gfCNCPoint3[10874] = {X 388.1959, Y 11.2433, Z -3.8333, A 0.000, B 0.000, C 0.000 }
gfCNCPoint3[10875] = {X 388.5095, Y 10.3472, Z -3.8333, A 0.000, B 0.000, C 0.000 }
gfCNCPoint3[10876] = {X 389.0147, Y 9.5432, Z -3.8333, A 0.000, B 0.000, C 0.000 }
gfCNCPoint3[10877] = {X 389.6860, Y 8.8719, Z -3.8333, A 0.000, B 0.000, C 0.000 }
gfCNCPoint3[10878] = {X 390.4900, Y 8.3667, Z -3.8333, A 0.000, B 0.000, C 0.000 }
gfCNCPoint3[10879] = {X 391.3861, Y 8.0531, Z -3.8333, A 0.000, B 0.000, C 0.000 }
gfCNCPoint3[10880] = {X 392.3296, Y 7.9468, Z -3.8333, A 0.000, B 0.000, C 0.000 }
gfCNCPoint3[10881] = {X 399.1118, Y 7.9468, Z -3.8333, A 0.000, B 0.000, C 0.000 }
gfCNCPoint3[10882] = {X 400.0552, Y 8.0531, Z -3.8333, A 0.000, B 0.000, C 0.000 }
gfCNCPoint3[10883] = {X 400.9514, Y 8.3667, Z -3.8333, A 0.000, B 0.000, C 0.000 }
gfCNCPoint3[10884] = {X 401.7554, Y 8.8718, Z -3.8333, A 0.000, B 0.000, C 0.000 }
gfCNCPoint3[10885] = {X 402.4267, Y 9.5432, Z -3.8333, A 0.000, B 0.000, C 0.000 }
gfCNCPoint3[10886] = {X 402.9319, Y 10.3471, Z -3.8333, A 0.000, B 0.000, C 0.000 }
gfCNCPoint3[10887] = {X 403.2455, Y 11.2433, Z -3.8333, A 0.000, B 0.000, C 0.000 }
gfCNCPoint3[10888] = {X 403.3518, Y 12.1868, Z -3.8333, A 0.000, B 0.000, C 0.000 }
gfCNCPoint3[10889] = {X 403.3518, Y 12.9781, Z -3.8333, A 0.000, B 0.000, C 0.000 }
gfCNCPoint3[10890] = {X 403.2466, Y 13.9164, Z -3.8333, A 0.000, B 0.000, C 0.000 }
gfCNCPoint3[10891] = {X 402.9365, Y 14.8081, Z -3.8333, A 0.000, B 0.000, C 0.000 }
gfCNCPoint3[10892] = {X 405.3544, Y 18.9789, Z -3.8333, A 0.000, B 0.000, C 0.000 }
gfCNCPoint3[10893] = {X 407.9641, Y 14.7597, Z -3.8333, A 0.000, B 0.000, C 0.000 }
gfCNCPoint3[10894] = {X 407.6748, Y 13.9080, Z -3.8333, A 0.000, B 0.000, C 0.000 }
gfCNCPoint3[10895] = {X 407.5717, Y 13.0144, Z -3.8333, A 0.000, B 0.000, C 0.000 }
gfCNCPoint3[10896] = {X 407.5715, Y 12.1868, Z -3.8333, A 0.000, B 0.000, C 0.000 }
gfCNCPoint3[10897] = {X 407.6778, Y 11.2433, Z -3.8333, A 0.000, B 0.000, C 0.000 }
gfCNCPoint3[10898] = {X 407.9914, Y 10.3471, Z -3.8333, A 0.000, B 0.000, C 0.000 }
gfCNCPoint3[10899] = {X 408.4966, Y 9.5432, Z -3.8333, A 0.000, B 0.000, C 0.000 }
gfCNCPoint3[10900] = {X 409.1679, Y 8.8718, Z -3.8333, A 0.000, B 0.000, C 0.000 }
gfCNCPoint3[10901] = {X 409.9719, Y 8.3667, Z -3.8333, A 0.000, B 0.000, C 0.000 }
gfCNCPoint3[10902] = {X 410.8680, Y 8.0531, Z -3.8333, A 0.000, B 0.000, C 0.000 }
gfCNCPoint3[10903] = {X 411.8115, Y 7.9468, Z -3.8333, A 0.000, B 0.000, C 0.000 }
gfCNCPoint3[10904] = {X 419.3245, Y 7.9468, Z -3.8333, A 0.000, B 0.000, C 0.000 }
gfCNCPoint3[10905] = {X 420.2679, Y 8.0531, Z -3.8333, A 0.000, B 0.000, C 0.000 }
gfCNCPoint3[10906] = {X 421.1641, Y 8.3667, Z -3.8333, A 0.000, B 0.000, C 0.000 }
gfCNCPoint3[10907] = {X 421.9681, Y 8.8718, Z -3.8333, A 0.000, B 0.000, C 0.000 }
gfCNCPoint3[10908] = {X 422.6394, Y 9.5432, Z -3.8333, A 0.000, B 0.000, C 0.000 }
gfCNCPoint3[10909] = {X 423.1446, Y 10.3471, Z -3.8333, A 0.000, B 0.000, C 0.000 }
gfCNCPoint3[10910] = {X 423.4582, Y 11.2433, Z -3.8333, A 0.000, B 0.000, C 0.000 }
gfCNCPoint3[10911] = {X 423.5645, Y 12.1868, Z -3.8333, A 0.000, B 0.000, C 0.000 }
gfCNCPoint3[10912] = {X 423.5645, Y 12.9798, Z -3.8333, A 0.000, B 0.000, C 0.000 }
gfCNCPoint3[10913] = {X 423.4723, Y 13.8340, Z -3.8333, A 0.000, B 0.000, C 0.000 }
gfCNCPoint3[10914] = {X 423.2124, Y 14.6529, Z -3.8333, A 0.000, B 0.000, C 0.000 }
gfCNCPoint3[10915] = {X 422.7950, Y 15.4039, Z -3.8333, A 0.000, B 0.000, C 0.000 }
gfCNCPoint3[10916] = {X 422.2368, Y 16.0570, Z -3.8333, A 0.000, B 0.000, C 0.000 }
gfCNCPoint3[10917] = {X 421.5600, Y 16.5863, Z -3.8333, A 0.000, B 0.000, C 0.000 }
gfCNCPoint3[10918] = {X 420.7916, Y 16.9706, Z -3.8333, A 0.000, B 0.000, C 0.000 }
gfCNCPoint3[10919] = {X 420.0648, Y 17.9463, Z -3.8333, A 0.000, B 0.000, C 0.000 }
gfCNCPoint3[10920] = {X 419.4075, Y 18.9700, Z -3.8333, A 0.000, B 0.000, C 0.000 }
gfCNCPoint3[10921] = {X 417.9262, Y 21.3685, Z -3.8333, A 0.000, B 0.000, C 0.000 }
gfCNCPoint3[10922] = {X 416.0825, Y 24.3294, Z -3.8333, A 0.000, B 0.000, C 0.000 }
gfCNCPoint3[10923] = {X 419.4780, Y 26.4437, Z -3.8333, A 0.000, B 0.000, C 0.000 }
gfCNCPoint3[10924] = {X 416.0146, Y 24.2871, Z -3.8333, A 0.000, B 0.000, C 0.000 }
gfCNCPoint3[10925] = {X 411.3866, Y 31.7193, Z -3.8333, A 0.000, B 0.000, C 0.000 }
gfCNCPoint3[10926] = {X 411.3873, Y 40.9718, Z -3.8333, A 0.000, B 0.000, C 0.000 }
gfCNCPoint3[10927] = {X 412.0246, Y 41.6368, Z -3.8333, A 0.000, B 0.000, C 0.000 }
gfCNCPoint3[10928] = {X 412.5050, Y 42.4226, Z -3.8333, A 0.000, B 0.000, C 0.000 }
gfCNCPoint3[10929] = {X 412.8064, Y 43.2930, Z -3.8333, A 0.000, B 0.000, C 0.000 }
gfCNCPoint3[10930] = {X 412.9147, Y 44.2077, Z -3.8333, A 0.000, B 0.000, C 0.000 }
gfCNCPoint3[10931] = {X 412.9147, Y 45.0002, Z -3.8333, A 0.000, B 0.000, C 0.000 }
gfCNCPoint3[10932] = {X 412.8103, Y 45.9258, Z -3.8333, A 0.000, B 0.000, C 0.000 }
gfCNCPoint3[10933] = {X 412.5027, Y 46.8051, Z -3.8333, A 0.000, B 0.000, C 0.000 }
gfCNCPoint3[10934] = {X 412.0070, Y 47.5938, Z -3.8333, A 0.000, B 0.000, C 0.000 }
gfCNCPoint3[10935] = {X 411.3483, Y 48.2525, Z -3.8333, A 0.000, B 0.000, C 0.000 }
gfCNCPoint3[10936] = {X 410.5596, Y 48.7480, Z -3.8333, A 0.000, B 0.000, C 0.000 }
gfCNCPoint3[10937] = {X 409.6803, Y 49.0557, Z -3.8333, A 0.000, B 0.000, C 0.000 }
gfCNCPoint3[10938] = {X 408.7547, Y 49.1600, Z -3.8333, A 0.000, B 0.000, C 0.000 }
gfCNCPoint3[10939] = {X 402.3112, Y 49.1600, Z -3.8333, A 0.000, B 0.000, C 0.000 }
gfCNCPoint3[10940] = {X 401.3900, Y 49.0567, Z -3.8333, A 0.000, B 0.000, C 0.000 }
gfCNCPoint3[10941] = {X 400.5146, Y 48.7520, Z -3.8333, A 0.000, B 0.000, C 0.000 }
gfCNCPoint3[10942] = {X 399.7283, Y 48.2610, Z -3.8333, A 0.000, B 0.000, C 0.000 }
gfCNCPoint3[10943] = {X 399.0703, Y 47.6081, Z -3.8333, A 0.000, B 0.000, C 0.000 }
gfCNCPoint3[10944] = {X 398.5732, Y 46.8257, Z -3.8333, A 0.000, B 0.000, C 0.000 }
gfCNCPoint3[10945] = {X 398.2617, Y 45.9526, Z -3.8333, A 0.000, B 0.000, C 0.000 }
gfCNCPoint3[10946] = {X 398.1513, Y 45.0322, Z -3.8333, A 0.000, B 0.000, C 0.000 }
gfCNCPoint3[10947] = {X 398.1516, Y 44.1549, Z -3.8333, A 0.000, B 0.000, C 0.000 }
gfCNCPoint3[10948] = {X 398.2616, Y 43.2570, Z -3.8333, A 0.000, B 0.000, C 0.000 }
gfCNCPoint3[10949] = {X 398.5630, Y 42.4041, Z -3.8333, A 0.000, B 0.000, C 0.000 }
gfCNCPoint3[10950] = {X 399.0417, Y 41.6366, Z -3.8333, A 0.000, B 0.000, C 0.000 }
gfCNCPoint3[10951] = {X 399.6750, Y 40.9907, Z -3.8333, A 0.000, B 0.000, C 0.000 }
gfCNCPoint3[10952] = {X 399.6327, Y 31.5567, Z -3.8333, A 0.000, B 0.000, C 0.000 }
gfCNCPoint3[10953] = {X 393.6516, Y 21.1559, Z -3.8333, A 0.000, B 0.000, C 0.000 }
gfCNCPoint3[10954] = {X 392.7632, Y 19.6448, Z -3.8333, A 0.000, B 0.000, C 0.000 }
gfCNCPoint3[10955] = {X 391.8461, Y 18.1509, Z -3.8333, A 0.000, B 0.000, C 0.000 }
gfCNCPoint3[10956] = {X 391.3435, Y 17.4543, Z -3.8333, A 0.000, B 0.000, C 0.000 }
gfCNCPoint3[10957] = {X 390.7552, Y 16.8286, Z -3.8333, A 0.000, B 0.000, C 0.000 }
gfCNCPoint3[10958] = {X 389.9030, Y 16.3569, Z -3.8333, A 0.000, B 0.000, C 0.000 }
gfCNCPoint3[10959] = {X 389.1838, Y 15.7000, Z -3.8333, A 0.000, B 0.000, C 0.000 }
gfCNCPoint3[10960] = {X 388.6371, Y 14.8939, Z -3.8333, A 0.000, B 0.000, C 0.000 }
gfCNCPoint3[10961] = {X 388.2928, Y 13.9828, Z -3.8333, A 0.000, B 0.000, C 0.000 }
gfCNCPoint3[10962] = {X 388.1698, Y 13.0166, Z -3.8333, A 0.000, B 0.000, C 0.000 }
gfCNCPoint3[10963] = {X 388.1696, Y 12.1868, Z -3.8333, A 0.000, B 0.000, C 0.000 }
gfCNCPoint3[10964] = {X 388.2739, Y 11.2611, Z -3.8333, A 0.000, B 0.000, C 0.000 }
gfCNCPoint3[10965] = {X 388.5816, Y 10.3819, Z -3.8333, A 0.000, B 0.000, C 0.000 }
gfCNCPoint3[10966] = {X 389.0772, Y 9.5931, Z -3.8333, A 0.000, B 0.000, C 0.000 }
gfCNCPoint3[10967] = {X 389.7359, Y 8.9344, Z -3.8333, A 0.000, B 0.000, C 0.000 }
gfCNCPoint3[10968] = {X 390.5247, Y 8.4388, Z -3.8333, A 0.000, B 0.000, C 0.000 }
gfCNCPoint3[10969] = {X 391.4039, Y 8.1311, Z -3.8333, A 0.000, B 0.000, C 0.000 }
gfCNCPoint3[10970] = {X 392.3296, Y 8.0268, Z -3.8333, A 0.000, B 0.000, C 0.000 }
gfCNCPoint3[10971] = {X 399.1118, Y 8.0268, Z -3.8333, A 0.000, B 0.000, C 0.000 }
gfCNCPoint3[10972] = {X 400.0374, Y 8.1311, Z -3.8333, A 0.000, B 0.000, C 0.000 }
gfCNCPoint3[10973] = {X 400.9167, Y 8.4388, Z -3.8333, A 0.000, B 0.000, C 0.000 }
gfCNCPoint3[10974] = {X 401.7055, Y 8.9344, Z -3.8333, A 0.000, B 0.000, C 0.000 }
gfCNCPoint3[10975] = {X 402.3642, Y 9.5931, Z -3.8333, A 0.000, B 0.000, C 0.000 }
gfCNCPoint3[10976] = {X 402.8598, Y 10.3819, Z -3.8333, A 0.000, B 0.000, C 0.000 }
gfCNCPoint3[10977] = {X 403.1675, Y 11.2611, Z -3.8333, A 0.000, B 0.000, C 0.000 }
gfCNCPoint3[10978] = {X 403.2718, Y 12.1868, Z -3.8333, A 0.000, B 0.000, C 0.000 }
gfCNCPoint3[10979] = {X 403.2718, Y 12.9781, Z -3.8333, A 0.000, B 0.000, C 0.000 }
gfCNCPoint3[10980] = {X 403.1639, Y 13.9192, Z -3.8333, A 0.000, B 0.000, C 0.000 }
gfCNCPoint3[10981] = {X 402.8459, Y 14.8115, Z -3.8333, A 0.000, B 0.000, C 0.000 }
gfCNCPoint3[10982] = {X 405.3522, Y 19.1346, Z -3.8333, A 0.000, B 0.000, C 0.000 }
gfCNCPoint3[10983] = {X 408.0549, Y 14.7650, Z -3.8333, A 0.000, B 0.000, C 0.000 }
gfCNCPoint3[10984] = {X 407.7576, Y 13.9114, Z -3.8333, A 0.000, B 0.000, C 0.000 }
gfCNCPoint3[10985] = {X 407.6517, Y 13.0137, Z -3.8333, A 0.000, B 0.000, C 0.000 }
gfCNCPoint3[10986] = {X 407.6515, Y 12.1868, Z -3.8333, A 0.000, B 0.000, C 0.000 }
gfCNCPoint3[10987] = {X 407.7558, Y 11.2611, Z -3.8333, A 0.000, B 0.000, C 0.000 }
gfCNCPoint3[10988] = {X 408.0635, Y 10.3819, Z -3.8333, A 0.000, B 0.000, C 0.000 }
gfCNCPoint3[10989] = {X 408.5591, Y 9.5931, Z -3.8333, A 0.000, B 0.000, C 0.000 }
gfCNCPoint3[10990] = {X 409.2178, Y 8.9344, Z -3.8333, A 0.000, B 0.000, C 0.000 }
gfCNCPoint3[10991] = {X 410.0066, Y 8.4388, Z -3.8333, A 0.000, B 0.000, C 0.000 }
gfCNCPoint3[10992] = {X 410.8859, Y 8.1311, Z -3.8333, A 0.000, B 0.000, C 0.000 }
gfCNCPoint3[10993] = {X 411.8115, Y 8.0268, Z -3.8333, A 0.000, B 0.000, C 0.000 }
gfCNCPoint3[10994] = {X 419.3245, Y 8.0268, Z -3.8333, A 0.000, B 0.000, C 0.000 }
gfCNCPoint3[10995] = {X 420.2501, Y 8.1311, Z -3.8333, A 0.000, B 0.000, C 0.000 }
gfCNCPoint3[10996] = {X 421.1294, Y 8.4388, Z -3.8333, A 0.000, B 0.000, C 0.000 }
gfCNCPoint3[10997] = {X 421.9182, Y 8.9344, Z -3.8333, A 0.000, B 0.000, C 0.000 }
gfCNCPoint3[10998] = {X 422.5769, Y 9.5931, Z -3.8333, A 0.000, B 0.000, C 0.000 }
gfCNCPoint3[10999] = {X 423.0725, Y 10.3819, Z -3.8333, A 0.000, B 0.000, C 0.000 }
gfCNCPoint3[11000] = {X 423.3802, Y 11.2611, Z -3.8333, A 0.000, B 0.000, C 0.000 }
gfCNCPoint3[11001] = {X 423.4845, Y 12.1868, Z -3.8333, A 0.000, B 0.000, C 0.000 }
gfCNCPoint3[11002] = {X 423.4845, Y 12.9792, Z -3.8333, A 0.000, B 0.000, C 0.000 }
gfCNCPoint3[11003] = {X 423.3933, Y 13.8210, Z -3.8333, A 0.000, B 0.000, C 0.000 }
gfCNCPoint3[11004] = {X 423.1361, Y 14.6278, Z -3.8333, A 0.000, B 0.000, C 0.000 }
gfCNCPoint3[11005] = {X 422.7231, Y 15.3671, Z -3.8333, A 0.000, B 0.000, C 0.000 }
gfCNCPoint3[11006] = {X 422.1710, Y 16.0092, Z -3.8333, A 0.000, B 0.000, C 0.000 }
gfCNCPoint3[11007] = {X 421.5020, Y 16.5283, Z -3.8333, A 0.000, B 0.000, C 0.000 }
gfCNCPoint3[11008] = {X 420.7429, Y 16.9035, Z -3.8333, A 0.000, B 0.000, C 0.000 }
gfCNCPoint3[11009] = {X 420.0054, Y 17.8914, Z -3.8333, A 0.000, B 0.000, C 0.000 }
gfCNCPoint3[11010] = {X 419.3390, Y 18.9286, Z -3.8333, A 0.000, B 0.000, C 0.000 }
gfCNCPoint3[11011] = {X 417.8583, Y 21.3264, Z -3.8333, A 0.000, B 0.000, C 0.000 }
gfCNCPoint3[11012] = {X 416.0146, Y 24.2871, Z -3.8333, A 0.000, B 0.000, C 0.000 }
gfCNCPoint3[11013] = {X 419.4101, Y 26.4014, Z -3.8333, A 0.000, B 0.000, C 0.000 }
gfCNCPoint3[11014] = {X 415.9467, Y 24.2448, Z -3.8333, A 0.000, B 0.000, C 0.000 }
gfCNCPoint3[11015] = {X 411.3066, Y 31.6964, Z -3.8333, A 0.000, B 0.000, C 0.000 }
gfCNCPoint3[11016] = {X 411.3073, Y 41.0093, Z -3.8333, A 0.000, B 0.000, C 0.000 }
gfCNCPoint3[11017] = {X 411.9442, Y 41.6636, Z -3.8333, A 0.000, B 0.000, C 0.000 }
gfCNCPoint3[11018] = {X 412.4247, Y 42.4400, Z -3.8333, A 0.000, B 0.000, C 0.000 }
gfCNCPoint3[11019] = {X 412.7263, Y 43.3018, Z -3.8333, A 0.000, B 0.000, C 0.000 }
gfCNCPoint3[11020] = {X 412.8347, Y 44.2085, Z -3.8333, A 0.000, B 0.000, C 0.000 }
gfCNCPoint3[11021] = {X 412.8347, Y 45.0002, Z -3.8333, A 0.000, B 0.000, C 0.000 }
gfCNCPoint3[11022] = {X 412.7324, Y 45.9080, Z -3.8333, A 0.000, B 0.000, C 0.000 }
gfCNCPoint3[11023] = {X 412.4306, Y 46.7703, Z -3.8333, A 0.000, B 0.000, C 0.000 }
gfCNCPoint3[11024] = {X 411.9445, Y 47.5439, Z -3.8333, A 0.000, B 0.000, C 0.000 }
gfCNCPoint3[11025] = {X 411.2985, Y 48.1899, Z -3.8333, A 0.000, B 0.000, C 0.000 }
gfCNCPoint3[11026] = {X 410.5249, Y 48.6760, Z -3.8333, A 0.000, B 0.000, C 0.000 }
gfCNCPoint3[11027] = {X 409.6625, Y 48.9777, Z -3.8333, A 0.000, B 0.000, C 0.000 }
gfCNCPoint3[11028] = {X 408.7547, Y 49.0800, Z -3.8333, A 0.000, B 0.000, C 0.000 }
gfCNCPoint3[11029] = {X 402.3112, Y 49.0800, Z -3.8333, A 0.000, B 0.000, C 0.000 }
gfCNCPoint3[11030] = {X 401.4077, Y 48.9787, Z -3.8333, A 0.000, B 0.000, C 0.000 }
gfCNCPoint3[11031] = {X 400.5491, Y 48.6799, Z -3.8333, A 0.000, B 0.000, C 0.000 }
gfCNCPoint3[11032] = {X 399.7780, Y 48.1983, Z -3.8333, A 0.000, B 0.000, C 0.000 }
gfCNCPoint3[11033] = {X 399.1326, Y 47.5579, Z -3.8333, A 0.000, B 0.000, C 0.000 }
gfCNCPoint3[11034] = {X 398.6451, Y 46.7906, Z -3.8333, A 0.000, B 0.000, C 0.000 }
gfCNCPoint3[11035] = {X 398.3396, Y 45.9343, Z -3.8333, A 0.000, B 0.000, C 0.000 }
gfCNCPoint3[11036] = {X 398.2313, Y 45.0316, Z -3.8333, A 0.000, B 0.000, C 0.000 }
gfCNCPoint3[11037] = {X 398.2316, Y 44.1559, Z -3.8333, A 0.000, B 0.000, C 0.000 }
gfCNCPoint3[11038] = {X 398.3416, Y 43.2661, Z -3.8333, A 0.000, B 0.000, C 0.000 }
gfCNCPoint3[11039] = {X 398.6434, Y 42.4218, Z -3.8333, A 0.000, B 0.000, C 0.000 }
gfCNCPoint3[11040] = {X 399.1223, Y 41.6638, Z -3.8333, A 0.000, B 0.000, C 0.000 }
gfCNCPoint3[11041] = {X 399.7552, Y 41.0287, Z -3.8333, A 0.000, B 0.000, C 0.000 }
gfCNCPoint3[11042] = {X 399.7126, Y 31.5351, Z -3.8333, A 0.000, B 0.000, C 0.000 }
gfCNCPoint3[11043] = {X 393.7210, Y 21.1161, Z -3.8333, A 0.000, B 0.000, C 0.000 }
gfCNCPoint3[11044] = {X 392.8318, Y 19.6036, Z -3.8333, A 0.000, B 0.000, C 0.000 }
gfCNCPoint3[11045] = {X 391.9139, Y 18.1084, Z -3.8333, A 0.000, B 0.000, C 0.000 }
gfCNCPoint3[11046] = {X 391.4005, Y 17.3977, Z -3.8333, A 0.000, B 0.000, C 0.000 }
gfCNCPoint3[11047] = {X 390.7990, Y 16.7600, Z -3.8333, A 0.000, B 0.000, C 0.000 }
gfCNCPoint3[11048] = {X 389.9591, Y 16.2987, Z -3.8333, A 0.000, B 0.000, C 0.000 }
gfCNCPoint3[11049] = {X 389.2500, Y 15.6543, Z -3.8333, A 0.000, B 0.000, C 0.000 }
gfCNCPoint3[11050] = {X 388.7108, Y 14.8623, Z -3.8333, A 0.000, B 0.000, C 0.000 }
gfCNCPoint3[11051] = {X 388.3711, Y 13.9663, Z -3.8333, A 0.000, B 0.000, C 0.000 }
gfCNCPoint3[11052] = {X 388.2498, Y 13.0158, Z -3.8333, A 0.000, B 0.000, C 0.000 }
gfCNCPoint3[11053] = {X 388.2496, Y 12.1868, Z -3.8333, A 0.000, B 0.000, C 0.000 }
gfCNCPoint3[11054] = {X 388.3519, Y 11.2789, Z -3.8333, A 0.000, B 0.000, C 0.000 }
gfCNCPoint3[11055] = {X 388.6537, Y 10.4166, Z -3.8333, A 0.000, B 0.000, C 0.000 }
gfCNCPoint3[11056] = {X 389.1398, Y 9.6430, Z -3.8333, A 0.000, B 0.000, C 0.000 }
gfCNCPoint3[11057] = {X 389.7858, Y 8.9969, Z -3.8333, A 0.000, B 0.000, C 0.000 }
gfCNCPoint3[11058] = {X 390.5594, Y 8.5109, Z -3.8333, A 0.000, B 0.000, C 0.000 }
gfCNCPoint3[11059] = {X 391.4217, Y 8.2091, Z -3.8333, A 0.000, B 0.000, C 0.000 }
gfCNCPoint3[11060] = {X 392.3296, Y 8.1068, Z -3.8333, A 0.000, B 0.000, C 0.000 }
gfCNCPoint3[11061] = {X 399.1118, Y 8.1068, Z -3.8333, A 0.000, B 0.000, C 0.000 }
gfCNCPoint3[11062] = {X 400.0196, Y 8.2091, Z -3.8333, A 0.000, B 0.000, C 0.000 }
gfCNCPoint3[11063] = {X 400.8820, Y 8.5109, Z -3.8333, A 0.000, B 0.000, C 0.000 }
gfCNCPoint3[11064] = {X 401.6556, Y 8.9969, Z -3.8333, A 0.000, B 0.000, C 0.000 }
gfCNCPoint3[11065] = {X 402.3016, Y 9.6430, Z -3.8333, A 0.000, B 0.000, C 0.000 }
gfCNCPoint3[11066] = {X 402.7877, Y 10.4166, Z -3.8333, A 0.000, B 0.000, C 0.000 }
gfCNCPoint3[11067] = {X 403.0895, Y 11.2789, Z -3.8333, A 0.000, B 0.000, C 0.000 }
gfCNCPoint3[11068] = {X 403.1918, Y 12.1868, Z -3.8333, A 0.000, B 0.000, C 0.000 }
gfCNCPoint3[11069] = {X 403.1918, Y 12.9781, Z -3.8333, A 0.000, B 0.000, C 0.000 }
gfCNCPoint3[11070] = {X 403.0811, Y 13.9219, Z -3.8333, A 0.000, B 0.000, C 0.000 }
gfCNCPoint3[11071] = {X 402.7551, Y 14.8144, Z -3.8333, A 0.000, B 0.000, C 0.000 }
gfCNCPoint3[11072] = {X 405.3499, Y 19.2903, Z -3.8333, A 0.000, B 0.000, C 0.000 }
gfCNCPoint3[11073] = {X 408.1460, Y 14.7697, Z -3.8333, A 0.000, B 0.000, C 0.000 }
gfCNCPoint3[11074] = {X 408.1093, Y 14.6926, Z -3.8333, A 0.000, B 0.000, C 0.000 }
gfCNCPoint3[11075] = {X 408.0742, Y 14.6147, Z -3.8333, A 0.000, B 0.000, C 0.000 }
gfCNCPoint3[11076] = {X 407.8218, Y 13.8313, Z -3.8333, A 0.000, B 0.000, C 0.000 }
gfCNCPoint3[11077] = {X 407.7317, Y 13.0131, Z -3.8333, A 0.000, B 0.000, C 0.000 }
gfCNCPoint3[11078] = {X 407.7315, Y 12.1868, Z -3.8333, A 0.000, B 0.000, C 0.000 }
gfCNCPoint3[11079] = {X 407.8338, Y 11.2789, Z -3.8333, A 0.000, B 0.000, C 0.000 }
gfCNCPoint3[11080] = {X 408.1356, Y 10.4166, Z -3.8333, A 0.000, B 0.000, C 0.000 }
gfCNCPoint3[11081] = {X 408.6217, Y 9.6430, Z -3.8333, A 0.000, B 0.000, C 0.000 }
gfCNCPoint3[11082] = {X 409.2677, Y 8.9969, Z -3.8333, A 0.000, B 0.000, C 0.000 }
gfCNCPoint3[11083] = {X 410.0413, Y 8.5109, Z -3.8333, A 0.000, B 0.000, C 0.000 }
gfCNCPoint3[11084] = {X 410.9037, Y 8.2091, Z -3.8333, A 0.000, B 0.000, C 0.000 }
gfCNCPoint3[11085] = {X 411.8115, Y 8.1068, Z -3.8333, A 0.000, B 0.000, C 0.000 }
gfCNCPoint3[11086] = {X 419.3245, Y 8.1068, Z -3.8333, A 0.000, B 0.000, C 0.000 }
gfCNCPoint3[11087] = {X 420.2323, Y 8.2091, Z -3.8333, A 0.000, B 0.000, C 0.000 }
gfCNCPoint3[11088] = {X 421.0947, Y 8.5109, Z -3.8333, A 0.000, B 0.000, C 0.000 }
gfCNCPoint3[11089] = {X 421.8683, Y 8.9969, Z -3.8333, A 0.000, B 0.000, C 0.000 }
gfCNCPoint3[11090] = {X 422.5143, Y 9.6430, Z -3.8333, A 0.000, B 0.000, C 0.000 }
gfCNCPoint3[11091] = {X 423.0004, Y 10.4166, Z -3.8333, A 0.000, B 0.000, C 0.000 }
gfCNCPoint3[11092] = {X 423.3022, Y 11.2789, Z -3.8333, A 0.000, B 0.000, C 0.000 }
gfCNCPoint3[11093] = {X 423.4045, Y 12.1868, Z -3.8333, A 0.000, B 0.000, C 0.000 }
gfCNCPoint3[11094] = {X 423.4045, Y 12.9786, Z -3.8333, A 0.000, B 0.000, C 0.000 }
gfCNCPoint3[11095] = {X 423.3143, Y 13.8081, Z -3.8333, A 0.000, B 0.000, C 0.000 }
gfCNCPoint3[11096] = {X 423.0598, Y 14.6027, Z -3.8333, A 0.000, B 0.000, C 0.000 }
gfCNCPoint3[11097] = {X 422.6513, Y 15.3302, Z -3.8333, A 0.000, B 0.000, C 0.000 }
gfCNCPoint3[11098] = {X 422.1053, Y 15.9612, Z -3.8333, A 0.000, B 0.000, C 0.000 }
gfCNCPoint3[11099] = {X 421.4441, Y 16.4701, Z -3.8333, A 0.000, B 0.000, C 0.000 }
gfCNCPoint3[11100] = {X 420.6943, Y 16.8362, Z -3.8333, A 0.000, B 0.000, C 0.000 }
gfCNCPoint3[11101] = {X 419.9462, Y 17.8365, Z -3.8333, A 0.000, B 0.000, C 0.000 }
gfCNCPoint3[11102] = {X 419.2706, Y 18.8871, Z -3.8333, A 0.000, B 0.000, C 0.000 }
gfCNCPoint3[11103] = {X 417.7903, Y 21.2842, Z -3.8333, A 0.000, B 0.000, C 0.000 }
gfCNCPoint3[11104] = {X 415.9467, Y 24.2448, Z -3.8333, A 0.000, B 0.000, C 0.000 }
gfCNCPoint3[11105] = {X 419.3422, Y 26.3592, Z -3.8333, A 0.000, B 0.000, C 0.000 }
gfCNCPoint3[11106] = {X 415.8788, Y 24.2025, Z -3.8333, A 0.000, B 0.000, C 0.000 }
gfCNCPoint3[11107] = {X 411.2266, Y 31.6735, Z -3.8333, A 0.000, B 0.000, C 0.000 }
gfCNCPoint3[11108] = {X 411.2273, Y 41.0472, Z -3.8333, A 0.000, B 0.000, C 0.000 }
gfCNCPoint3[11109] = {X 411.8636, Y 41.6906, Z -3.8333, A 0.000, B 0.000, C 0.000 }
gfCNCPoint3[11110] = {X 412.3443, Y 42.4574, Z -3.8333, A 0.000, B 0.000, C 0.000 }
gfCNCPoint3[11111] = {X 412.6462, Y 43.3105, Z -3.8333, A 0.000, B 0.000, C 0.000 }
gfCNCPoint3[11112] = {X 412.7547, Y 44.2089, Z -3.8333, A 0.000, B 0.000, C 0.000 }
gfCNCPoint3[11113] = {X 412.7545, Y 45.0384, Z -3.8333, A 0.000, B 0.000, C 0.000 }
gfCNCPoint3[11114] = {X 412.6469, Y 45.9222, Z -3.8333, A 0.000, B 0.000, C 0.000 }
gfCNCPoint3[11115] = {X 412.3466, Y 46.7602, Z -3.8333, A 0.000, B 0.000, C 0.000 }
gfCNCPoint3[11116] = {X 411.8683, Y 47.5111, Z -3.8333, A 0.000, B 0.000, C 0.000 }
gfCNCPoint3[11117] = {X 411.2357, Y 48.1376, Z -3.8333, A 0.000, B 0.000, C 0.000 }
gfCNCPoint3[11118] = {X 410.4803, Y 48.6086, Z -3.8333, A 0.000, B 0.000, C 0.000 }
gfCNCPoint3[11119] = {X 409.6394, Y 48.9009, Z -3.8333, A 0.000, B 0.000, C 0.000 }
gfCNCPoint3[11120] = {X 408.7547, Y 49.0000, Z -3.8333, A 0.000, B 0.000, C 0.000 }
gfCNCPoint3[11121] = {X 402.3112, Y 49.0000, Z -3.8333, A 0.000, B 0.000, C 0.000 }
gfCNCPoint3[11122] = {X 401.4211, Y 48.8997, Z -3.8333, A 0.000, B 0.000, C 0.000 }
gfCNCPoint3[11123] = {X 400.5757, Y 48.6039, Z -3.8333, A 0.000, B 0.000, C 0.000 }
gfCNCPoint3[11124] = {X 399.8172, Y 48.1273, Z -3.8333, A 0.000, B 0.000, C 0.000 }
gfCNCPoint3[11125] = {X 399.1839, Y 47.4939, Z -3.8333, A 0.000, B 0.000, C 0.000 }
gfCNCPoint3[11126] = {X 398.7073, Y 46.7355, Z -3.8333, A 0.000, B 0.000, C 0.000 }
gfCNCPoint3[11127] = {X 398.4115, Y 45.8900, Z -3.8333, A 0.000, B 0.000, C 0.000 }
gfCNCPoint3[11128] = {X 398.3112, Y 45.0000, Z -3.8333, A 0.000, B 0.000, C 0.000 }
gfCNCPoint3[11129] = {X 398.3115, Y 44.1569, Z -3.8333, A 0.000, B 0.000, C 0.000 }
gfCNCPoint3[11130] = {X 398.4217, Y 43.2753, Z -3.8333, A 0.000, B 0.000, C 0.000 }
gfCNCPoint3[11131] = {X 398.7237, Y 42.4397, Z -3.8333, A 0.000, B 0.000, C 0.000 }
gfCNCPoint3[11132] = {X 399.2028, Y 41.6913, Z -3.8333, A 0.000, B 0.000, C 0.000 }
gfCNCPoint3[11133] = {X 399.8352, Y 41.0672, Z -3.8333, A 0.000, B 0.000, C 0.000 }
gfCNCPoint3[11134] = {X 399.8376, Y 31.5921, Z -3.8333, A 0.000, B 0.000, C 0.000 }
gfCNCPoint3[11135] = {X 393.7903, Y 21.0762, Z -3.8333, A 0.000, B 0.000, C 0.000 }
gfCNCPoint3[11136] = {X 392.9004, Y 19.5624, Z -3.8333, A 0.000, B 0.000, C 0.000 }
gfCNCPoint3[11137] = {X 391.9816, Y 18.0659, Z -3.8333, A 0.000, B 0.000, C 0.000 }
gfCNCPoint3[11138] = {X 391.4575, Y 17.3410, Z -3.8333, A 0.000, B 0.000, C 0.000 }
gfCNCPoint3[11139] = {X 390.8426, Y 16.6913, Z -3.8333, A 0.000, B 0.000, C 0.000 }
gfCNCPoint3[11140] = {X 390.0091, Y 16.2361, Z -3.8333, A 0.000, B 0.000, C 0.000 }
gfCNCPoint3[11141] = {X 389.3064, Y 15.5972, Z -3.8333, A 0.000, B 0.000, C 0.000 }
gfCNCPoint3[11142] = {X 388.7742, Y 14.8107, Z -3.8333, A 0.000, B 0.000, C 0.000 }
gfCNCPoint3[11143] = {X 388.4423, Y 13.9209, Z -3.8333, A 0.000, B 0.000, C 0.000 }
gfCNCPoint3[11144] = {X 388.3296, Y 12.9779, Z -3.8333, A 0.000, B 0.000, C 0.000 }
gfCNCPoint3[11145] = {X 388.3296, Y 12.1868, Z -3.8333, A 0.000, B 0.000, C 0.000 }
gfCNCPoint3[11146] = {X 388.4299, Y 11.2967, Z -3.8333, A 0.000, B 0.000, C 0.000 }
gfCNCPoint3[11147] = {X 388.7258, Y 10.4513, Z -3.8333, A 0.000, B 0.000, C 0.000 }
gfCNCPoint3[11148] = {X 389.2023, Y 9.6929, Z -3.8333, A 0.000, B 0.000, C 0.000 }
gfCNCPoint3[11149] = {X 389.8357, Y 9.0595, Z -3.8333, A 0.000, B 0.000, C 0.000 }
gfCNCPoint3[11150] = {X 390.5941, Y 8.5829, Z -3.8333, A 0.000, B 0.000, C 0.000 }
gfCNCPoint3[11151] = {X 391.4395, Y 8.2871, Z -3.8333, A 0.000, B 0.000, C 0.000 }
gfCNCPoint3[11152] = {X 392.3296, Y 8.1868, Z -3.8333, A 0.000, B 0.000, C 0.000 }
gfCNCPoint3[11153] = {X 399.1118, Y 8.1868, Z -3.8333, A 0.000, B 0.000, C 0.000 }
gfCNCPoint3[11154] = {X 400.0018, Y 8.2871, Z -3.8333, A 0.000, B 0.000, C 0.000 }
gfCNCPoint3[11155] = {X 400.8473, Y 8.5829, Z -3.8333, A 0.000, B 0.000, C 0.000 }
gfCNCPoint3[11156] = {X 401.6057, Y 9.0595, Z -3.8333, A 0.000, B 0.000, C 0.000 }
gfCNCPoint3[11157] = {X 402.2391, Y 9.6929, Z -3.8333, A 0.000, B 0.000, C 0.000 }
gfCNCPoint3[11158] = {X 402.7156, Y 10.4513, Z -3.8333, A 0.000, B 0.000, C 0.000 }
gfCNCPoint3[11159] = {X 403.0115, Y 11.2967, Z -3.8333, A 0.000, B 0.000, C 0.000 }
gfCNCPoint3[11160] = {X 403.1118, Y 12.1868, Z -3.8333, A 0.000, B 0.000, C 0.000 }
gfCNCPoint3[11161] = {X 403.1115, Y 13.0192, Z -3.8333, A 0.000, B 0.000, C 0.000 }
gfCNCPoint3[11162] = {X 402.9933, Y 13.9442, Z -3.8333, A 0.000, B 0.000, C 0.000 }
gfCNCPoint3[11163] = {X 402.6641, Y 14.8167, Z -3.8333, A 0.000, B 0.000, C 0.000 }
gfCNCPoint3[11164] = {X 405.2576, Y 19.3199, Z -3.8333, A 0.000, B 0.000, C 0.000 }
gfCNCPoint3[11165] = {X 405.3712, Y 19.4080, Z -3.8333, A 0.000, B 0.000, C 0.000 }
gfCNCPoint3[11166] = {X 408.1949, Y 14.8342, Z -3.8333, A 0.000, B 0.000, C 0.000 }
gfCNCPoint3[11167] = {X 408.2428, Y 14.7847, Z -3.8333, A 0.000, B 0.000, C 0.000 }
gfCNCPoint3[11168] = {X 408.1937, Y 14.6843, Z -3.8333, A 0.000, B 0.000, C 0.000 }
gfCNCPoint3[11169] = {X 408.1475, Y 14.5826, Z -3.8333, A 0.000, B 0.000, C 0.000 }
gfCNCPoint3[11170] = {X 407.8964, Y 13.7977, Z -3.8333, A 0.000, B 0.000, C 0.000 }
gfCNCPoint3[11171] = {X 407.8115, Y 12.9779, Z -3.8333, A 0.000, B 0.000, C 0.000 }
gfCNCPoint3[11172] = {X 407.8115, Y 12.1868, Z -3.8333, A 0.000, B 0.000, C 0.000 }
gfCNCPoint3[11173] = {X 407.9118, Y 11.2967, Z -3.8333, A 0.000, B 0.000, C 0.000 }
gfCNCPoint3[11174] = {X 408.2077, Y 10.4513, Z -3.8333, A 0.000, B 0.000, C 0.000 }
gfCNCPoint3[11175] = {X 408.6842, Y 9.6929, Z -3.8333, A 0.000, B 0.000, C 0.000 }
gfCNCPoint3[11176] = {X 409.3176, Y 9.0595, Z -3.8333, A 0.000, B 0.000, C 0.000 }
gfCNCPoint3[11177] = {X 410.0760, Y 8.5829, Z -3.8333, A 0.000, B 0.000, C 0.000 }
gfCNCPoint3[11178] = {X 410.9215, Y 8.2871, Z -3.8333, A 0.000, B 0.000, C 0.000 }
gfCNCPoint3[11179] = {X 411.8115, Y 8.1868, Z -3.8333, A 0.000, B 0.000, C 0.000 }
gfCNCPoint3[11180] = {X 419.3245, Y 8.1868, Z -3.8333, A 0.000, B 0.000, C 0.000 }
gfCNCPoint3[11181] = {X 420.2145, Y 8.2871, Z -3.8333, A 0.000, B 0.000, C 0.000 }
gfCNCPoint3[11182] = {X 421.0600, Y 8.5829, Z -3.8333, A 0.000, B 0.000, C 0.000 }
gfCNCPoint3[11183] = {X 421.8184, Y 9.0595, Z -3.8333, A 0.000, B 0.000, C 0.000 }
gfCNCPoint3[11184] = {X 422.4518, Y 9.6929, Z -3.8333, A 0.000, B 0.000, C 0.000 }
gfCNCPoint3[11185] = {X 422.9283, Y 10.4513, Z -3.8333, A 0.000, B 0.000, C 0.000 }
gfCNCPoint3[11186] = {X 423.2242, Y 11.2967, Z -3.8333, A 0.000, B 0.000, C 0.000 }
gfCNCPoint3[11187] = {X 423.3245, Y 12.1868, Z -3.8333, A 0.000, B 0.000, C 0.000 }
gfCNCPoint3[11188] = {X 423.3245, Y 12.9780, Z -3.8333, A 0.000, B 0.000, C 0.000 }
gfCNCPoint3[11189] = {X 423.1977, Y 13.9553, Z -3.8333, A 0.000, B 0.000, C 0.000 }
gfCNCPoint3[11190] = {X 422.8393, Y 14.8735, Z -3.8333, A 0.000, B 0.000, C 0.000 }
gfCNCPoint3[11191] = {X 422.2706, Y 15.6784, Z -3.8333, A 0.000, B 0.000, C 0.000 }
gfCNCPoint3[11192] = {X 421.5249, Y 16.3228, Z -3.8333, A 0.000, B 0.000, C 0.000 }
gfCNCPoint3[11193] = {X 420.6460, Y 16.7687, Z -3.8333, A 0.000, B 0.000, C 0.000 }
gfCNCPoint3[11194] = {X 419.8870, Y 17.7815, Z -3.8333, A 0.000, B 0.000, C 0.000 }
gfCNCPoint3[11195] = {X 419.2022, Y 18.8457, Z -3.8333, A 0.000, B 0.000, C 0.000 }
gfCNCPoint3[11196] = {X 417.7223, Y 21.2420, Z -3.8333, A 0.000, B 0.000, C 0.000 }
gfCNCPoint3[11197] = {X 415.8788, Y 24.2025, Z -3.8333, A 0.000, B 0.000, C 0.000 }
gfCNCPoint3[11198] = {X 419.3422, Y 26.3592, Z -3.8333, A 0.000, B 0.000, C 0.000 }
gfCNCPoint3[11199] = {X 419.3422, Y 26.3592, Z -0.8333, A 0.000, B 0.000, C 0.000 }
gfCNCPoint3[11200] = {X 419.3422, Y 26.3592, Z 11.0000, A 0.000, B 0.000, C 0.000 }
gfCNCPoint3[11201] = {X 352.3320, Y -3.5327, Z 11.0000, A 0.000, B 0.000, C 0.000 }
gfCNCPoint3[11202] = {X 352.3320, Y -3.5327, Z -0.8333, A 0.000, B 0.000, C 0.000 }
gfCNCPoint3[11203] = {X 352.3320, Y -3.5327, Z -3.8333, A 0.000, B 0.000, C 0.000 }
gfCNCPoint3[11204] = {X 351.5861, Y 0.4785, Z -3.8333, A 0.000, B 0.000, C 0.000 }
gfCNCPoint3[11205] = {X 351.8696, Y 0.5313, Z -3.8333, A 0.000, B 0.000, C 0.000 }
gfCNCPoint3[11206] = {X 353.8045, Y 1.0172, Z -3.8333, A 0.000, B 0.000, C 0.000 }
gfCNCPoint3[11207] = {X 355.6846, Y 1.6844, Z -3.8333, A 0.000, B 0.000, C 0.000 }
gfCNCPoint3[11208] = {X 357.4930, Y 2.5269, Z -3.8333, A 0.000, B 0.000, C 0.000 }
gfCNCPoint3[11209] = {X 359.2134, Y 3.5369, Z -3.8333, A 0.000, B 0.000, C 0.000 }
gfCNCPoint3[11210] = {X 360.8303, Y 4.7055, Z -3.8333, A 0.000, B 0.000, C 0.000 }
gfCNCPoint3[11211] = {X 362.3292, Y 6.0221, Z -3.8333, A 0.000, B 0.000, C 0.000 }
gfCNCPoint3[11212] = {X 363.6965, Y 7.4749, Z -3.8333, A 0.000, B 0.000, C 0.000 }
gfCNCPoint3[11213] = {X 365.1623, Y 9.3666, Z -3.8333, A 0.000, B 0.000, C 0.000 }
gfCNCPoint3[11214] = {X 366.4383, Y 11.3913, Z -3.8333, A 0.000, B 0.000, C 0.000 }
gfCNCPoint3[11215] = {X 367.5125, Y 13.5298, Z -3.8333, A 0.000, B 0.000, C 0.000 }
gfCNCPoint3[11216] = {X 368.3749, Y 15.7623, Z -3.8333, A 0.000, B 0.000, C 0.000 }
gfCNCPoint3[11217] = {X 369.0174, Y 18.0676, Z -3.8333, A 0.000, B 0.000, C 0.000 }
gfCNCPoint3[11218] = {X 369.4997, Y 20.7039, Z -3.8333, A 0.000, B 0.000, C 0.000 }
gfCNCPoint3[11219] = {X 369.7570, Y 23.3717, Z -3.8333, A 0.000, B 0.000, C 0.000 }
gfCNCPoint3[11220] = {X 369.7875, Y 26.0516, Z -3.8333, A 0.000, B 0.000, C 0.000 }
gfCNCPoint3[11221] = {X 369.5909, Y 28.7245, Z -3.8333, A 0.000, B 0.000, C 0.000 }
gfCNCPoint3[11222] = {X 369.1687, Y 31.3711, Z -3.8333, A 0.000, B 0.000, C 0.000 }
gfCNCPoint3[11223] = {X 368.6448, Y 33.4754, Z -3.8333, A 0.000, B 0.000, C 0.000 }
gfCNCPoint3[11224] = {X 367.9371, Y 35.5252, Z -3.8333, A 0.000, B 0.000, C 0.000 }
gfCNCPoint3[11225] = {X 367.0510, Y 37.5044, Z -3.8333, A 0.000, B 0.000, C 0.000 }
gfCNCPoint3[11226] = {X 365.9935, Y 39.3976, Z -3.8333, A 0.000, B 0.000, C 0.000 }
gfCNCPoint3[11227] = {X 364.7729, Y 41.1900, Z -3.8333, A 0.000, B 0.000, C 0.000 }
gfCNCPoint3[11228] = {X 364.6545, Y 41.3524, Z -3.8333, A 0.000, B 0.000, C 0.000 }
gfCNCPoint3[11229] = {X 364.0232, Y 42.1276, Z -3.8333, A 0.000, B 0.000, C 0.000 }
gfCNCPoint3[11230] = {X 362.7624, Y 43.5421, Z -3.8333, A 0.000, B 0.000, C 0.000 }
gfCNCPoint3[11231] = {X 361.3808, Y 44.8389, Z -3.8333, A 0.000, B 0.000, C 0.000 }
gfCNCPoint3[11232] = {X 359.8894, Y 46.0078, Z -3.8333, A 0.000, B 0.000, C 0.000 }
gfCNCPoint3[11233] = {X 358.3000, Y 47.0395, Z -3.8333, A 0.000, B 0.000, C 0.000 }
gfCNCPoint3[11234] = {X 356.6252, Y 47.9258, Z -3.8333, A 0.000, B 0.000, C 0.000 }
gfCNCPoint3[11235] = {X 356.2220, Y 48.1167, Z -3.8333, A 0.000, B 0.000, C 0.000 }
gfCNCPoint3[11236] = {X 354.0243, Y 48.9372, Z -3.8333, A 0.000, B 0.000, C 0.000 }
gfCNCPoint3[11237] = {X 351.7544, Y 49.5297, Z -3.8333, A 0.000, B 0.000, C 0.000 }
gfCNCPoint3[11238] = {X 349.4361, Y 49.8881, Z -3.8333, A 0.000, B 0.000, C 0.000 }
gfCNCPoint3[11239] = {X 347.0933, Y 50.0086, Z -3.8333, A 0.000, B 0.000, C 0.000 }
gfCNCPoint3[11240] = {X 345.0267, Y 49.9738, Z -3.8333, A 0.000, B 0.000, C 0.000 }
gfCNCPoint3[11241] = {X 342.9709, Y 49.7598, Z -3.8333, A 0.000, B 0.000, C 0.000 }
gfCNCPoint3[11242] = {X 340.9414, Y 49.3684, Z -3.8333, A 0.000, B 0.000, C 0.000 }
gfCNCPoint3[11243] = {X 338.9535, Y 48.8024, Z -3.8333, A 0.000, B 0.000, C 0.000 }
gfCNCPoint3[11244] = {X 337.0222, Y 48.0661, Z -3.8333, A 0.000, B 0.000, C 0.000 }
gfCNCPoint3[11245] = {X 335.1621, Y 47.1650, Z -3.8333, A 0.000, B 0.000, C 0.000 }
gfCNCPoint3[11246] = {X 333.5780, Y 46.1875, Z -3.8333, A 0.000, B 0.000, C 0.000 }
gfCNCPoint3[11247] = {X 332.0750, Y 45.0892, Z -3.8333, A 0.000, B 0.000, C 0.000 }
gfCNCPoint3[11248] = {X 330.6624, Y 43.8770, Z -3.8333, A 0.000, B 0.000, C 0.000 }
gfCNCPoint3[11249] = {X 329.7213, Y 43.8764, Z -3.8333, A 0.000, B 0.000, C 0.000 }
gfCNCPoint3[11250] = {X 328.8027, Y 43.6721, Z -3.8333, A 0.000, B 0.000, C 0.000 }
gfCNCPoint3[11251] = {X 327.9501, Y 43.2738, Z -3.8333, A 0.000, B 0.000, C 0.000 }
gfCNCPoint3[11252] = {X 327.2040, Y 42.7002, Z -3.8333, A 0.000, B 0.000, C 0.000 }
gfCNCPoint3[11253] = {X 326.5808, Y 42.0925, Z -3.8333, A 0.000, B 0.000, C 0.000 }
gfCNCPoint3[11254] = {X 325.9523, Y 41.3190, Z -3.8333, A 0.000, B 0.000, C 0.000 }
gfCNCPoint3[11255] = {X 325.5179, Y 40.4220, Z -3.8333, A 0.000, B 0.000, C 0.000 }
gfCNCPoint3[11256] = {X 325.3006, Y 39.4493, Z -3.8333, A 0.000, B 0.000, C 0.000 }
gfCNCPoint3[11257] = {X 325.3120, Y 38.4527, Z -3.8333, A 0.000, B 0.000, C 0.000 }
gfCNCPoint3[11258] = {X 325.5514, Y 37.4852, Z -3.8333, A 0.000, B 0.000, C 0.000 }
gfCNCPoint3[11259] = {X 326.0062, Y 36.5984, Z -3.8333, A 0.000, B 0.000, C 0.000 }
gfCNCPoint3[11260] = {X 330.2395, Y 30.2687, Z -3.8333, A 0.000, B 0.000, C 0.000 }
gfCNCPoint3[11261] = {X 330.8409, Y 29.5518, Z -3.8333, A 0.000, B 0.000, C 0.000 }
gfCNCPoint3[11262] = {X 331.5826, Y 28.9812, Z -3.8333, A 0.000, B 0.000, C 0.000 }
gfCNCPoint3[11263] = {X 332.4297, Y 28.5837, Z -3.8333, A 0.000, B 0.000, C 0.000 }
gfCNCPoint3[11264] = {X 333.3425, Y 28.3780, Z -3.8333, A 0.000, B 0.000, C 0.000 }
gfCNCPoint3[11265] = {X 334.2782, Y 28.3736, Z -3.8333, A 0.000, B 0.000, C 0.000 }
gfCNCPoint3[11266] = {X 335.1929, Y 28.5708, Z -3.8333, A 0.000, B 0.000, C 0.000 }
gfCNCPoint3[11267] = {X 336.0437, Y 28.9604, Z -3.8333, A 0.000, B 0.000, C 0.000 }
gfCNCPoint3[11268] = {X 336.7907, Y 29.5240, Z -3.8333, A 0.000, B 0.000, C 0.000 }
gfCNCPoint3[11269] = {X 337.4284, Y 30.1382, Z -3.8333, A 0.000, B 0.000, C 0.000 }
gfCNCPoint3[11270] = {X 337.9530, Y 30.7612, Z -3.8333, A 0.000, B 0.000, C 0.000 }
gfCNCPoint3[11271] = {X 338.3513, Y 31.4717, Z -3.8333, A 0.000, B 0.000, C 0.000 }
gfCNCPoint3[11272] = {X 338.6092, Y 32.2442, Z -3.8333, A 0.000, B 0.000, C 0.000 }
gfCNCPoint3[11273] = {X 338.7175, Y 33.0514, Z -3.8333, A 0.000, B 0.000, C 0.000 }
gfCNCPoint3[11274] = {X 338.6724, Y 33.8646, Z -3.8333, A 0.000, B 0.000, C 0.000 }
gfCNCPoint3[11275] = {X 339.4360, Y 34.5560, Z -3.8333, A 0.000, B 0.000, C 0.000 }
gfCNCPoint3[11276] = {X 340.2334, Y 35.2080, Z -3.8333, A 0.000, B 0.000, C 0.000 }
gfCNCPoint3[11277] = {X 341.5307, Y 36.0601, Z -3.8333, A 0.000, B 0.000, C 0.000 }
gfCNCPoint3[11278] = {X 342.9384, Y 36.7138, Z -3.8333, A 0.000, B 0.000, C 0.000 }
gfCNCPoint3[11279] = {X 344.4264, Y 37.1554, Z -3.8333, A 0.000, B 0.000, C 0.000 }
gfCNCPoint3[11280] = {X 345.9629, Y 37.3752, Z -3.8333, A 0.000, B 0.000, C 0.000 }
gfCNCPoint3[11281] = {X 347.5150, Y 37.3686, Z -3.8333, A 0.000, B 0.000, C 0.000 }
gfCNCPoint3[11282] = {X 348.9558, Y 37.1756, Z -3.8333, A 0.000, B 0.000, C 0.000 }
gfCNCPoint3[11283] = {X 350.3459, Y 36.7506, Z -3.8333, A 0.000, B 0.000, C 0.000 }
gfCNCPoint3[11284] = {X 351.6482, Y 36.1048, Z -3.8333, A 0.000, B 0.000, C 0.000 }
gfCNCPoint3[11285] = {X 352.8280, Y 35.2555, Z -3.8333, A 0.000, B 0.000, C 0.000 }
gfCNCPoint3[11286] = {X 353.9819, Y 34.1346, Z -3.8333, A 0.000, B 0.000, C 0.000 }
gfCNCPoint3[11287] = {X 354.9806, Y 32.8734, Z -3.8333, A 0.000, B 0.000, C 0.000 }
gfCNCPoint3[11288] = {X 355.8070, Y 31.4932, Z -3.8333, A 0.000, B 0.000, C 0.000 }
gfCNCPoint3[11289] = {X 356.4473, Y 30.0174, Z -3.8333, A 0.000, B 0.000, C 0.000 }
gfCNCPoint3[11290] = {X 356.8905, Y 28.4710, Z -3.8333, A 0.000, B 0.000, C 0.000 }
gfCNCPoint3[11291] = {X 357.1638, Y 26.7828, Z -3.8333, A 0.000, B 0.000, C 0.000 }
gfCNCPoint3[11292] = {X 357.2751, Y 25.0762, Z -3.8333, A 0.000, B 0.000, C 0.000 }
gfCNCPoint3[11293] = {X 357.2234, Y 23.3668, Z -3.8333, A 0.000, B 0.000, C 0.000 }
gfCNCPoint3[11294] = {X 357.0092, Y 21.6701, Z -3.8333, A 0.000, B 0.000, C 0.000 }
gfCNCPoint3[11295] = {X 356.6730, Y 20.2205, Z -3.8333, A 0.000, B 0.000, C 0.000 }
gfCNCPoint3[11296] = {X 356.1600, Y 18.8237, Z -3.8333, A 0.000, B 0.000, C 0.000 }
gfCNCPoint3[11297] = {X 355.4780, Y 17.5012, Z -3.8333, A 0.000, B 0.000, C 0.000 }
gfCNCPoint3[11298] = {X 354.6376, Y 16.2732, Z -3.8333, A 0.000, B 0.000, C 0.000 }
gfCNCPoint3[11299] = {X 353.7517, Y 15.2852, Z -3.8333, A 0.000, B 0.000, C 0.000 }
gfCNCPoint3[11300] = {X 352.7334, Y 14.4343, Z -3.8333, A 0.000, B 0.000, C 0.000 }
gfCNCPoint3[11301] = {X 351.6037, Y 13.7381, Z -3.8333, A 0.000, B 0.000, C 0.000 }
gfCNCPoint3[11302] = {X 350.3860, Y 13.2109, Z -3.8333, A 0.000, B 0.000, C 0.000 }
gfCNCPoint3[11303] = {X 349.1052, Y 12.8636, Z -3.8333, A 0.000, B 0.000, C 0.000 }
gfCNCPoint3[11304] = {X 347.3449, Y 12.6448, Z -3.8333, A 0.000, B 0.000, C 0.000 }
gfCNCPoint3[11305] = {X 345.5711, Y 12.6607, Z -3.8333, A 0.000, B 0.000, C 0.000 }
gfCNCPoint3[11306] = {X 343.8149, Y 12.9110, Z -3.8333, A 0.000, B 0.000, C 0.000 }
gfCNCPoint3[11307] = {X 342.1073, Y 13.3914, Z -3.8333, A 0.000, B 0.000, C 0.000 }
gfCNCPoint3[11308] = {X 340.4782, Y 14.0935, Z -3.8333, A 0.000, B 0.000, C 0.000 }
gfCNCPoint3[11309] = {X 338.9564, Y 15.0049, Z -3.8333, A 0.000, B 0.000, C 0.000 }
gfCNCPoint3[11310] = {X 338.9176, Y 15.8496, Z -3.8333, A 0.000, B 0.000, C 0.000 }
gfCNCPoint3[11311] = {X 338.7150, Y 16.6707, Z -3.8333, A 0.000, B 0.000, C 0.000 }
gfCNCPoint3[11312] = {X 338.3563, Y 17.4365, Z -3.8333, A 0.000, B 0.000, C 0.000 }
gfCNCPoint3[11313] = {X 337.8553, Y 18.1178, Z -3.8333, A 0.000, B 0.000, C 0.000 }
gfCNCPoint3[11314] = {X 337.2312, Y 18.6884, Z -3.8333, A 0.000, B 0.000, C 0.000 }
gfCNCPoint3[11315] = {X 336.5140, Y 19.2162, Z -3.8333, A 0.000, B 0.000, C 0.000 }
gfCNCPoint3[11316] = {X 335.6982, Y 19.6754, Z -3.8333, A 0.000, B 0.000, C 0.000 }
gfCNCPoint3[11317] = {X 334.8027, Y 19.9480, Z -3.8333, A 0.000, B 0.000, C 0.000 }
gfCNCPoint3[11318] = {X 333.8694, Y 20.0213, Z -3.8333, A 0.000, B 0.000, C 0.000 }
gfCNCPoint3[11319] = {X 332.9422, Y 19.8919, Z -3.8333, A 0.000, B 0.000, C 0.000 }
gfCNCPoint3[11320] = {X 332.0647, Y 19.5657, Z -3.8333, A 0.000, B 0.000, C 0.000 }
gfCNCPoint3[11321] = {X 331.2781, Y 19.0582, Z -3.8333, A 0.000, B 0.000, C 0.000 }
gfCNCPoint3[11322] = {X 330.6193, Y 18.3931, Z -3.8333, A 0.000, B 0.000, C 0.000 }
gfCNCPoint3[11323] = {X 330.1192, Y 17.6017, Z -3.8333, A 0.000, B 0.000, C 0.000 }
gfCNCPoint3[11324] = {X 326.5942, Y 10.3502, Z -3.8333, A 0.000, B 0.000, C 0.000 }
gfCNCPoint3[11325] = {X 326.2930, Y 9.5271, Z -3.8333, A 0.000, B 0.000, C 0.000 }
gfCNCPoint3[11326] = {X 326.1640, Y 8.6602, Z -3.8333, A 0.000, B 0.000, C 0.000 }
gfCNCPoint3[11327] = {X 326.2128, Y 7.7851, Z -3.8333, A 0.000, B 0.000, C 0.000 }
gfCNCPoint3[11328] = {X 326.4371, Y 6.9378, Z -3.8333, A 0.000, B 0.000, C 0.000 }
gfCNCPoint3[11329] = {X 326.8279, Y 6.1532, Z -3.8333, A 0.000, B 0.000, C 0.000 }
gfCNCPoint3[11330] = {X 327.3690, Y 5.4637, Z -3.8333, A 0.000, B 0.000, C 0.000 }
gfCNCPoint3[11331] = {X 328.0381, Y 4.8976, Z -3.8333, A 0.000, B 0.000, C 0.000 }
gfCNCPoint3[11332] = {X 328.7084, Y 4.4385, Z -3.8333, A 0.000, B 0.000, C 0.000 }
gfCNCPoint3[11333] = {X 329.5889, Y 3.9825, Z -3.8333, A 0.000, B 0.000, C 0.000 }
gfCNCPoint3[11334] = {X 330.5501, Y 3.7393, Z -3.8333, A 0.000, B 0.000, C 0.000 }
gfCNCPoint3[11335] = {X 331.5415, Y 3.7217, Z -3.8333, A 0.000, B 0.000, C 0.000 }
gfCNCPoint3[11336] = {X 332.5109, Y 3.9305, Z -3.8333, A 0.000, B 0.000, C 0.000 }
gfCNCPoint3[11337] = {X 333.9976, Y 3.1009, Z -3.8333, A 0.000, B 0.000, C 0.000 }
gfCNCPoint3[11338] = {X 335.5315, Y 2.3619, Z -3.8333, A 0.000, B 0.000, C 0.000 }
gfCNCPoint3[11339] = {X 337.6677, Y 1.4953, Z -3.8333, A 0.000, B 0.000, C 0.000 }
gfCNCPoint3[11340] = {X 339.8716, Y 0.8193, Z -3.8333, A 0.000, B 0.000, C 0.000 }
gfCNCPoint3[11341] = {X 342.1263, Y 0.3390, Z -3.8333, A 0.000, B 0.000, C 0.000 }
gfCNCPoint3[11342] = {X 344.4143, Y 0.0581, Z -3.8333, A 0.000, B 0.000, C 0.000 }
gfCNCPoint3[11343] = {X 346.7182, Y -0.0212, Z -3.8333, A 0.000, B 0.000, C 0.000 }
gfCNCPoint3[11344] = {X 349.0202, Y 0.1017, Z -3.8333, A 0.000, B 0.000, C 0.000 }
gfCNCPoint3[11345] = {X 351.3026, Y 0.4258, Z -3.8333, A 0.000, B 0.000, C 0.000 }
gfCNCPoint3[11346] = {X 351.5861, Y 0.4785, Z -3.8333, A 0.000, B 0.000, C 0.000 }
gfCNCPoint3[11347] = {X 352.3174, Y -3.4540, Z -3.8333, A 0.000, B 0.000, C 0.000 }
gfCNCPoint3[11348] = {X 351.5715, Y 0.5572, Z -3.8333, A 0.000, B 0.000, C 0.000 }
gfCNCPoint3[11349] = {X 351.8544, Y 0.6098, Z -3.8333, A 0.000, B 0.000, C 0.000 }
gfCNCPoint3[11350] = {X 353.7818, Y 1.0940, Z -3.8333, A 0.000, B 0.000, C 0.000 }
gfCNCPoint3[11351] = {X 355.6547, Y 1.7586, Z -3.8333, A 0.000, B 0.000, C 0.000 }
gfCNCPoint3[11352] = {X 357.4561, Y 2.5979, Z -3.8333, A 0.000, B 0.000, C 0.000 }
gfCNCPoint3[11353] = {X 359.1699, Y 3.6041, Z -3.8333, A 0.000, B 0.000, C 0.000 }
gfCNCPoint3[11354] = {X 360.7806, Y 4.7682, Z -3.8333, A 0.000, B 0.000, C 0.000 }
gfCNCPoint3[11355] = {X 362.2736, Y 6.0797, Z -3.8333, A 0.000, B 0.000, C 0.000 }
gfCNCPoint3[11356] = {X 363.6357, Y 7.5269, Z -3.8333, A 0.000, B 0.000, C 0.000 }
gfCNCPoint3[11357] = {X 365.0967, Y 9.4125, Z -3.8333, A 0.000, B 0.000, C 0.000 }
gfCNCPoint3[11358] = {X 366.3686, Y 11.4306, Z -3.8333, A 0.000, B 0.000, C 0.000 }
gfCNCPoint3[11359] = {X 367.4394, Y 13.5622, Z -3.8333, A 0.000, B 0.000, C 0.000 }
gfCNCPoint3[11360] = {X 368.2990, Y 15.7874, Z -3.8333, A 0.000, B 0.000, C 0.000 }
gfCNCPoint3[11361] = {X 368.9393, Y 18.0853, Z -3.8333, A 0.000, B 0.000, C 0.000 }
gfCNCPoint3[11362] = {X 369.4205, Y 20.7150, Z -3.8333, A 0.000, B 0.000, C 0.000 }
gfCNCPoint3[11363] = {X 369.6771, Y 23.3760, Z -3.8333, A 0.000, B 0.000, C 0.000 }
gfCNCPoint3[11364] = {X 369.7075, Y 26.0491, Z -3.8333, A 0.000, B 0.000, C 0.000 }
gfCNCPoint3[11365] = {X 369.5115, Y 28.7152, Z -3.8333, A 0.000, B 0.000, C 0.000 }
gfCNCPoint3[11366] = {X 369.0903, Y 31.3552, Z -3.8333, A 0.000, B 0.000, C 0.000 }
gfCNCPoint3[11367] = {X 368.5681, Y 33.4527, Z -3.8333, A 0.000, B 0.000, C 0.000 }
gfCNCPoint3[11368] = {X 367.8626, Y 35.4959, Z -3.8333, A 0.000, B 0.000, C 0.000 }
gfCNCPoint3[11369] = {X 366.9794, Y 37.4688, Z -3.8333, A 0.000, B 0.000, C 0.000 }
gfCNCPoint3[11370] = {X 365.9253, Y 39.3559, Z -3.8333, A 0.000, B 0.000, C 0.000 }
gfCNCPoint3[11371] = {X 364.7086, Y 41.1425, Z -3.8333, A 0.000, B 0.000, C 0.000 }
gfCNCPoint3[11372] = {X 364.5912, Y 41.3036, Z -3.8333, A 0.000, B 0.000, C 0.000 }
gfCNCPoint3[11373] = {X 363.9612, Y 42.0770, Z -3.8333, A 0.000, B 0.000, C 0.000 }
gfCNCPoint3[11374] = {X 362.7051, Y 43.4862, Z -3.8333, A 0.000, B 0.000, C 0.000 }
gfCNCPoint3[11375] = {X 361.3287, Y 44.7782, Z -3.8333, A 0.000, B 0.000, C 0.000 }
gfCNCPoint3[11376] = {X 359.8429, Y 45.9427, Z -3.8333, A 0.000, B 0.000, C 0.000 }
gfCNCPoint3[11377] = {X 358.2595, Y 46.9705, Z -3.8333, A 0.000, B 0.000, C 0.000 }
gfCNCPoint3[11378] = {X 356.5910, Y 47.8535, Z -3.8333, A 0.000, B 0.000, C 0.000 }
gfCNCPoint3[11379] = {X 356.1902, Y 48.0433, Z -3.8333, A 0.000, B 0.000, C 0.000 }
gfCNCPoint3[11380] = {X 353.9999, Y 48.8610, Z -3.8333, A 0.000, B 0.000, C 0.000 }
gfCNCPoint3[11381] = {X 351.7377, Y 49.4515, Z -3.8333, A 0.000, B 0.000, C 0.000 }
gfCNCPoint3[11382] = {X 349.4271, Y 49.8086, Z -3.8333, A 0.000, B 0.000, C 0.000 }
gfCNCPoint3[11383] = {X 347.0922, Y 49.9286, Z -3.8333, A 0.000, B 0.000, C 0.000 }
gfCNCPoint3[11384] = {X 345.0325, Y 49.8940, Z -3.8333, A 0.000, B 0.000, C 0.000 }
gfCNCPoint3[11385] = {X 342.9836, Y 49.6808, Z -3.8333, A 0.000, B 0.000, C 0.000 }
gfCNCPoint3[11386] = {X 340.9608, Y 49.2908, Z -3.8333, A 0.000, B 0.000, C 0.000 }
gfCNCPoint3[11387] = {X 338.9796, Y 48.7267, Z -3.8333, A 0.000, B 0.000, C 0.000 }
gfCNCPoint3[11388] = {X 337.0547, Y 47.9929, Z -3.8333, A 0.000, B 0.000, C 0.000 }
gfCNCPoint3[11389] = {X 335.2007, Y 47.0950, Z -3.8333, A 0.000, B 0.000, C 0.000 }
gfCNCPoint3[11390] = {X 333.6120, Y 46.1140, Z -3.8333, A 0.000, B 0.000, C 0.000 }
gfCNCPoint3[11391] = {X 332.1053, Y 45.0112, Z -3.8333, A 0.000, B 0.000, C 0.000 }
gfCNCPoint3[11392] = {X 330.6899, Y 43.7933, Z -3.8333, A 0.000, B 0.000, C 0.000 }
gfCNCPoint3[11393] = {X 329.7573, Y 43.7998, Z -3.8333, A 0.000, B 0.000, C 0.000 }
gfCNCPoint3[11394] = {X 328.8457, Y 43.6022, Z -3.8333, A 0.000, B 0.000, C 0.000 }
gfCNCPoint3[11395] = {X 327.9994, Y 43.2101, Z -3.8333, A 0.000, B 0.000, C 0.000 }
gfCNCPoint3[11396] = {X 327.2594, Y 42.6425, Z -3.8333, A 0.000, B 0.000, C 0.000 }
gfCNCPoint3[11397] = {X 326.6366, Y 42.0352, Z -3.8333, A 0.000, B 0.000, C 0.000 }
gfCNCPoint3[11398] = {X 326.0198, Y 41.2760, Z -3.8333, A 0.000, B 0.000, C 0.000 }
gfCNCPoint3[11399] = {X 325.5934, Y 40.3956, Z -3.8333, A 0.000, B 0.000, C 0.000 }
gfCNCPoint3[11400] = {X 325.3802, Y 39.4410, Z -3.8333, A 0.000, B 0.000, C 0.000 }
gfCNCPoint3[11401] = {X 325.3913, Y 38.4628, Z -3.8333, A 0.000, B 0.000, C 0.000 }
gfCNCPoint3[11402] = {X 325.6264, Y 37.5133, Z -3.8333, A 0.000, B 0.000, C 0.000 }
gfCNCPoint3[11403] = {X 326.0727, Y 36.6429, Z -3.8333, A 0.000, B 0.000, C 0.000 }
gfCNCPoint3[11404] = {X 330.3060, Y 30.3132, Z -3.8333, A 0.000, B 0.000, C 0.000 }
gfCNCPoint3[11405] = {X 330.8963, Y 29.6096, Z -3.8333, A 0.000, B 0.000, C 0.000 }
gfCNCPoint3[11406] = {X 331.6242, Y 29.0495, Z -3.8333, A 0.000, B 0.000, C 0.000 }
gfCNCPoint3[11407] = {X 332.4556, Y 28.6594, Z -3.8333, A 0.000, B 0.000, C 0.000 }
gfCNCPoint3[11408] = {X 333.3515, Y 28.4575, Z -3.8333, A 0.000, B 0.000, C 0.000 }
gfCNCPoint3[11409] = {X 334.2699, Y 28.4532, Z -3.8333, A 0.000, B 0.000, C 0.000 }
gfCNCPoint3[11410] = {X 335.1677, Y 28.6467, Z -3.8333, A 0.000, B 0.000, C 0.000 }
gfCNCPoint3[11411] = {X 336.0027, Y 29.0291, Z -3.8333, A 0.000, B 0.000, C 0.000 }
gfCNCPoint3[11412] = {X 336.7358, Y 29.5823, Z -3.8333, A 0.000, B 0.000, C 0.000 }
gfCNCPoint3[11413] = {X 337.3723, Y 30.1953, Z -3.8333, A 0.000, B 0.000, C 0.000 }
gfCNCPoint3[11414] = {X 337.8919, Y 30.8136, Z -3.8333, A 0.000, B 0.000, C 0.000 }
gfCNCPoint3[11415] = {X 338.2848, Y 31.5192, Z -3.8333, A 0.000, B 0.000, C 0.000 }
gfCNCPoint3[11416] = {X 338.5368, Y 32.2865, Z -3.8333, A 0.000, B 0.000, C 0.000 }
gfCNCPoint3[11417] = {X 338.6387, Y 33.0877, Z -3.8333, A 0.000, B 0.000, C 0.000 }
gfCNCPoint3[11418] = {X 338.5869, Y 33.8936, Z -3.8333, A 0.000, B 0.000, C 0.000 }
gfCNCPoint3[11419] = {X 339.3680, Y 34.6031, Z -3.8333, A 0.000, B 0.000, C 0.000 }
gfCNCPoint3[11420] = {X 340.1845, Y 35.2713, Z -3.8333, A 0.000, B 0.000, C 0.000 }
gfCNCPoint3[11421] = {X 341.4915, Y 36.1298, Z -3.8333, A 0.000, B 0.000, C 0.000 }
gfCNCPoint3[11422] = {X 342.9096, Y 36.7885, Z -3.8333, A 0.000, B 0.000, C 0.000 }
gfCNCPoint3[11423] = {X 344.4086, Y 37.2334, Z -3.8333, A 0.000, B 0.000, C 0.000 }
gfCNCPoint3[11424] = {X 345.9565, Y 37.4549, Z -3.8333, A 0.000, B 0.000, C 0.000 }
gfCNCPoint3[11425] = {X 347.5201, Y 37.4485, Z -3.8333, A 0.000, B 0.000, C 0.000 }
gfCNCPoint3[11426] = {X 348.9736, Y 37.2536, Z -3.8333, A 0.000, B 0.000, C 0.000 }
gfCNCPoint3[11427] = {X 350.3759, Y 36.8247, Z -3.8333, A 0.000, B 0.000, C 0.000 }
gfCNCPoint3[11428] = {X 351.6897, Y 36.1732, Z -3.8333, A 0.000, B 0.000, C 0.000 }
gfCNCPoint3[11429] = {X 352.8799, Y 35.3164, Z -3.8333, A 0.000, B 0.000, C 0.000 }
gfCNCPoint3[11430] = {X 354.0413, Y 34.1882, Z -3.8333, A 0.000, B 0.000, C 0.000 }
gfCNCPoint3[11431] = {X 355.0465, Y 32.9188, Z -3.8333, A 0.000, B 0.000, C 0.000 }
gfCNCPoint3[11432] = {X 355.8783, Y 31.5297, Z -3.8333, A 0.000, B 0.000, C 0.000 }
gfCNCPoint3[11433] = {X 356.5227, Y 30.0443, Z -3.8333, A 0.000, B 0.000, C 0.000 }
gfCNCPoint3[11434] = {X 356.9687, Y 28.4878, Z -3.8333, A 0.000, B 0.000, C 0.000 }
gfCNCPoint3[11435] = {X 357.2432, Y 26.7920, Z -3.8333, A 0.000, B 0.000, C 0.000 }
gfCNCPoint3[11436] = {X 357.3551, Y 25.0778, Z -3.8333, A 0.000, B 0.000, C 0.000 }
gfCNCPoint3[11437] = {X 357.3032, Y 23.3607, Z -3.8333, A 0.000, B 0.000, C 0.000 }
gfCNCPoint3[11438] = {X 357.0880, Y 21.6563, Z -3.8333, A 0.000, B 0.000, C 0.000 }
gfCNCPoint3[11439] = {X 356.7496, Y 20.1972, Z -3.8333, A 0.000, B 0.000, C 0.000 }
gfCNCPoint3[11440] = {X 356.2331, Y 18.7913, Z -3.8333, A 0.000, B 0.000, C 0.000 }
gfCNCPoint3[11441] = {X 355.5466, Y 17.4600, Z -3.8333, A 0.000, B 0.000, C 0.000 }
gfCNCPoint3[11442] = {X 354.7006, Y 16.2240, Z -3.8333, A 0.000, B 0.000, C 0.000 }
gfCNCPoint3[11443] = {X 353.8071, Y 15.2275, Z -3.8333, A 0.000, B 0.000, C 0.000 }
gfCNCPoint3[11444] = {X 352.7800, Y 14.3693, Z -3.8333, A 0.000, B 0.000, C 0.000 }
gfCNCPoint3[11445] = {X 351.6406, Y 13.6671, Z -3.8333, A 0.000, B 0.000, C 0.000 }
gfCNCPoint3[11446] = {X 350.4123, Y 13.1354, Z -3.8333, A 0.000, B 0.000, C 0.000 }
gfCNCPoint3[11447] = {X 349.1205, Y 12.7851, Z -3.8333, A 0.000, B 0.000, C 0.000 }
gfCNCPoint3[11448] = {X 347.3421, Y 12.5645, Z -3.8333, A 0.000, B 0.000, C 0.000 }
gfCNCPoint3[11449] = {X 345.5502, Y 12.5820, Z -3.8333, A 0.000, B 0.000, C 0.000 }
gfCNCPoint3[11450] = {X 343.7765, Y 12.8374, Z -3.8333, A 0.000, B 0.000, C 0.000 }
gfCNCPoint3[11451] = {X 342.0524, Y 13.3261, Z -3.8333, A 0.000, B 0.000, C 0.000 }
gfCNCPoint3[11452] = {X 340.4085, Y 14.0394, Z -3.8333, A 0.000, B 0.000, C 0.000 }
gfCNCPoint3[11453] = {X 338.8739, Y 14.9648, Z -3.8333, A 0.000, B 0.000, C 0.000 }
gfCNCPoint3[11454] = {X 338.8434, Y 15.8030, Z -3.8333, A 0.000, B 0.000, C 0.000 }
gfCNCPoint3[11455] = {X 338.6484, Y 16.6189, Z -3.8333, A 0.000, B 0.000, C 0.000 }
gfCNCPoint3[11456] = {X 338.2966, Y 17.3804, Z -3.8333, A 0.000, B 0.000, C 0.000 }
gfCNCPoint3[11457] = {X 337.8017, Y 18.0577, Z -3.8333, A 0.000, B 0.000, C 0.000 }
gfCNCPoint3[11458] = {X 337.1833, Y 18.6244, Z -3.8333, A 0.000, B 0.000, C 0.000 }
gfCNCPoint3[11459] = {X 336.4675, Y 19.1512, Z -3.8333, A 0.000, B 0.000, C 0.000 }
gfCNCPoint3[11460] = {X 335.6668, Y 19.6018, Z -3.8333, A 0.000, B 0.000, C 0.000 }
gfCNCPoint3[11461] = {X 334.7878, Y 19.8694, Z -3.8333, A 0.000, B 0.000, C 0.000 }
gfCNCPoint3[11462] = {X 333.8718, Y 19.9414, Z -3.8333, A 0.000, B 0.000, C 0.000 }
gfCNCPoint3[11463] = {X 332.9618, Y 19.8143, Z -3.8333, A 0.000, B 0.000, C 0.000 }
gfCNCPoint3[11464] = {X 332.1006, Y 19.4942, Z -3.8333, A 0.000, B 0.000, C 0.000 }
gfCNCPoint3[11465] = {X 331.3285, Y 18.9960, Z -3.8333, A 0.000, B 0.000, C 0.000 }
gfCNCPoint3[11466] = {X 330.6819, Y 18.3433, Z -3.8333, A 0.000, B 0.000, C 0.000 }
gfCNCPoint3[11467] = {X 330.1911, Y 17.5665, Z -3.8333, A 0.000, B 0.000, C 0.000 }
gfCNCPoint3[11468] = {X 326.6662, Y 10.3152, Z -3.8333, A 0.000, B 0.000, C 0.000 }
gfCNCPoint3[11469] = {X 326.3374, Y 9.3676, Z -3.8333, A 0.000, B 0.000, C 0.000 }
gfCNCPoint3[11470] = {X 326.2405, Y 8.3693, Z -3.8333, A 0.000, B 0.000, C 0.000 }
gfCNCPoint3[11471] = {X 326.3807, Y 7.3762, Z -3.8333, A 0.000, B 0.000, C 0.000 }
gfCNCPoint3[11472] = {X 326.7504, Y 6.4438, Z -3.8333, A 0.000, B 0.000, C 0.000 }
gfCNCPoint3[11473] = {X 327.3287, Y 5.6243, Z -3.8333, A 0.000, B 0.000, C 0.000 }
gfCNCPoint3[11474] = {X 328.0833, Y 4.9636, Z -3.8333, A 0.000, B 0.000, C 0.000 }
gfCNCPoint3[11475] = {X 328.7533, Y 4.5047, Z -3.8333, A 0.000, B 0.000, C 0.000 }
gfCNCPoint3[11476] = {X 329.6261, Y 4.0540, Z -3.8333, A 0.000, B 0.000, C 0.000 }
gfCNCPoint3[11477] = {X 330.5792, Y 3.8162, Z -3.8333, A 0.000, B 0.000, C 0.000 }
gfCNCPoint3[11478] = {X 331.5614, Y 3.8041, Z -3.8333, A 0.000, B 0.000, C 0.000 }
gfCNCPoint3[11479] = {X 332.5200, Y 4.0183, Z -3.8333, A 0.000, B 0.000, C 0.000 }
gfCNCPoint3[11480] = {X 334.0182, Y 3.1803, Z -3.8333, A 0.000, B 0.000, C 0.000 }
gfCNCPoint3[11481] = {X 335.5645, Y 2.4348, Z -3.8333, A 0.000, B 0.000, C 0.000 }
gfCNCPoint3[11482] = {X 337.6942, Y 1.5708, Z -3.8333, A 0.000, B 0.000, C 0.000 }
gfCNCPoint3[11483] = {X 339.8915, Y 0.8968, Z -3.8333, A 0.000, B 0.000, C 0.000 }
gfCNCPoint3[11484] = {X 342.1393, Y 0.4179, Z -3.8333, A 0.000, B 0.000, C 0.000 }
gfCNCPoint3[11485] = {X 344.4205, Y 0.1378, Z -3.8333, A 0.000, B 0.000, C 0.000 }
gfCNCPoint3[11486] = {X 346.7174, Y 0.0588, Z -3.8333, A 0.000, B 0.000, C 0.000 }
gfCNCPoint3[11487] = {X 349.0125, Y 0.1813, Z -3.8333, A 0.000, B 0.000, C 0.000 }
gfCNCPoint3[11488] = {X 351.2879, Y 0.5045, Z -3.8333, A 0.000, B 0.000, C 0.000 }
gfCNCPoint3[11489] = {X 351.5715, Y 0.5572, Z -3.8333, A 0.000, B 0.000, C 0.000 }
gfCNCPoint3[11490] = {X 352.3028, Y -3.3754, Z -3.8333, A 0.000, B 0.000, C 0.000 }
gfCNCPoint3[11491] = {X 351.5568, Y 0.6358, Z -3.8333, A 0.000, B 0.000, C 0.000 }
gfCNCPoint3[11492] = {X 351.8392, Y 0.6883, Z -3.8333, A 0.000, B 0.000, C 0.000 }
gfCNCPoint3[11493] = {X 353.7592, Y 1.1707, Z -3.8333, A 0.000, B 0.000, C 0.000 }
gfCNCPoint3[11494] = {X 355.6248, Y 1.8328, Z -3.8333, A 0.000, B 0.000, C 0.000 }
gfCNCPoint3[11495] = {X 357.4192, Y 2.6688, Z -3.8333, A 0.000, B 0.000, C 0.000 }
gfCNCPoint3[11496] = {X 359.1264, Y 3.6712, Z -3.8333, A 0.000, B 0.000, C 0.000 }
gfCNCPoint3[11497] = {X 360.7308, Y 4.8308, Z -3.8333, A 0.000, B 0.000, C 0.000 }
gfCNCPoint3[11498] = {X 362.2181, Y 6.1373, Z -3.8333, A 0.000, B 0.000, C 0.000 }
gfCNCPoint3[11499] = {X 363.5749, Y 7.5789, Z -3.8333, A 0.000, B 0.000, C 0.000 }
gfCNCPoint3[11500] = {X 365.0312, Y 9.4584, Z -3.8333, A 0.000, B 0.000, C 0.000 }
gfCNCPoint3[11501] = {X 366.2990, Y 11.4699, Z -3.8333, A 0.000, B 0.000, C 0.000 }
gfCNCPoint3[11502] = {X 367.3662, Y 13.5946, Z -3.8333, A 0.000, B 0.000, C 0.000 }
gfCNCPoint3[11503] = {X 368.2230, Y 15.8126, Z -3.8333, A 0.000, B 0.000, C 0.000 }
gfCNCPoint3[11504] = {X 368.8613, Y 18.1030, Z -3.8333, A 0.000, B 0.000, C 0.000 }
gfCNCPoint3[11505] = {X 369.3412, Y 20.7260, Z -3.8333, A 0.000, B 0.000, C 0.000 }
gfCNCPoint3[11506] = {X 369.5973, Y 23.3803, Z -3.8333, A 0.000, B 0.000, C 0.000 }
gfCNCPoint3[11507] = {X 369.6276, Y 26.0466, Z -3.8333, A 0.000, B 0.000, C 0.000 }
gfCNCPoint3[11508] = {X 369.4320, Y 28.7060, Z -3.8333, A 0.000, B 0.000, C 0.000 }
gfCNCPoint3[11509] = {X 369.0119, Y 31.3392, Z -3.8333, A 0.000, B 0.000, C 0.000 }
gfCNCPoint3[11510] = {X 368.4914, Y 33.4300, Z -3.8333, A 0.000, B 0.000, C 0.000 }
gfCNCPoint3[11511] = {X 367.7882, Y 35.4666, Z -3.8333, A 0.000, B 0.000, C 0.000 }
gfCNCPoint3[11512] = {X 366.9078, Y 37.4331, Z -3.8333, A 0.000, B 0.000, C 0.000 }
gfCNCPoint3[11513] = {X 365.8571, Y 39.3141, Z -3.8333, A 0.000, B 0.000, C 0.000 }
gfCNCPoint3[11514] = {X 364.6443, Y 41.0949, Z -3.8333, A 0.000, B 0.000, C 0.000 }
gfCNCPoint3[11515] = {X 364.5278, Y 41.2547, Z -3.8333, A 0.000, B 0.000, C 0.000 }
gfCNCPoint3[11516] = {X 363.8991, Y 42.0265, Z -3.8333, A 0.000, B 0.000, C 0.000 }
gfCNCPoint3[11517] = {X 362.6478, Y 43.4304, Z -3.8333, A 0.000, B 0.000, C 0.000 }
gfCNCPoint3[11518] = {X 361.2766, Y 44.7175, Z -3.8333, A 0.000, B 0.000, C 0.000 }
gfCNCPoint3[11519] = {X 359.7964, Y 45.8776, Z -3.8333, A 0.000, B 0.000, C 0.000 }
gfCNCPoint3[11520] = {X 358.2190, Y 46.9015, Z -3.8333, A 0.000, B 0.000, C 0.000 }
gfCNCPoint3[11521] = {X 356.5567, Y 47.7812, Z -3.8333, A 0.000, B 0.000, C 0.000 }
gfCNCPoint3[11522] = {X 356.1572, Y 47.9704, Z -3.8333, A 0.000, B 0.000, C 0.000 }
gfCNCPoint3[11523] = {X 353.9745, Y 48.7851, Z -3.8333, A 0.000, B 0.000, C 0.000 }
gfCNCPoint3[11524] = {X 351.7203, Y 49.3734, Z -3.8333, A 0.000, B 0.000, C 0.000 }
gfCNCPoint3[11525] = {X 349.4178, Y 49.7291, Z -3.8333, A 0.000, B 0.000, C 0.000 }
gfCNCPoint3[11526] = {X 347.0911, Y 49.8486, Z -3.8333, A 0.000, B 0.000, C 0.000 }
gfCNCPoint3[11527] = {X 345.0383, Y 49.8142, Z -3.8333, A 0.000, B 0.000, C 0.000 }
gfCNCPoint3[11528] = {X 342.9962, Y 49.6018, Z -3.8333, A 0.000, B 0.000, C 0.000 }
gfCNCPoint3[11529] = {X 340.9803, Y 49.2131, Z -3.8333, A 0.000, B 0.000, C 0.000 }
gfCNCPoint3[11530] = {X 339.0056, Y 48.6511, Z -3.8333, A 0.000, B 0.000, C 0.000 }
gfCNCPoint3[11531] = {X 337.0872, Y 47.9198, Z -3.8333, A 0.000, B 0.000, C 0.000 }
gfCNCPoint3[11532] = {X 335.2394, Y 47.0249, Z -3.8333, A 0.000, B 0.000, C 0.000 }
gfCNCPoint3[11533] = {X 333.6460, Y 46.0404, Z -3.8333, A 0.000, B 0.000, C 0.000 }
gfCNCPoint3[11534] = {X 332.1355, Y 44.9329, Z -3.8333, A 0.000, B 0.000, C 0.000 }
gfCNCPoint3[11535] = {X 330.7172, Y 43.7094, Z -3.8333, A 0.000, B 0.000, C 0.000 }
gfCNCPoint3[11536] = {X 329.7931, Y 43.7230, Z -3.8333, A 0.000, B 0.000, C 0.000 }
gfCNCPoint3[11537] = {X 328.8887, Y 43.5322, Z -3.8333, A 0.000, B 0.000, C 0.000 }
gfCNCPoint3[11538] = {X 328.0488, Y 43.1465, Z -3.8333, A 0.000, B 0.000, C 0.000 }
gfCNCPoint3[11539] = {X 327.3148, Y 42.5847, Z -3.8333, A 0.000, B 0.000, C 0.000 }
gfCNCPoint3[11540] = {X 326.6925, Y 41.9780, Z -3.8333, A 0.000, B 0.000, C 0.000 }
gfCNCPoint3[11541] = {X 326.0873, Y 41.2331, Z -3.8333, A 0.000, B 0.000, C 0.000 }
gfCNCPoint3[11542] = {X 325.6690, Y 40.3693, Z -3.8333, A 0.000, B 0.000, C 0.000 }
gfCNCPoint3[11543] = {X 325.4597, Y 39.4326, Z -3.8333, A 0.000, B 0.000, C 0.000 }
gfCNCPoint3[11544] = {X 325.4707, Y 38.4730, Z -3.8333, A 0.000, B 0.000, C 0.000 }
gfCNCPoint3[11545] = {X 325.7013, Y 37.5413, Z -3.8333, A 0.000, B 0.000, C 0.000 }
gfCNCPoint3[11546] = {X 326.1392, Y 36.6874, Z -3.8333, A 0.000, B 0.000, C 0.000 }
gfCNCPoint3[11547] = {X 330.3725, Y 30.3577, Z -3.8333, A 0.000, B 0.000, C 0.000 }
gfCNCPoint3[11548] = {X 330.9516, Y 29.6673, Z -3.8333, A 0.000, B 0.000, C 0.000 }
gfCNCPoint3[11549] = {X 331.6658, Y 29.1179, Z -3.8333, A 0.000, B 0.000, C 0.000 }
gfCNCPoint3[11550] = {X 332.4815, Y 28.7351, Z -3.8333, A 0.000, B 0.000, C 0.000 }
gfCNCPoint3[11551] = {X 333.3606, Y 28.5370, Z -3.8333, A 0.000, B 0.000, C 0.000 }
gfCNCPoint3[11552] = {X 334.2616, Y 28.5327, Z -3.8333, A 0.000, B 0.000, C 0.000 }
gfCNCPoint3[11553] = {X 335.1425, Y 28.7226, Z -3.8333, A 0.000, B 0.000, C 0.000 }
gfCNCPoint3[11554] = {X 335.9617, Y 29.0978, Z -3.8333, A 0.000, B 0.000, C 0.000 }
gfCNCPoint3[11555] = {X 336.6810, Y 29.6405, Z -3.8333, A 0.000, B 0.000, C 0.000 }
gfCNCPoint3[11556] = {X 337.3163, Y 30.2523, Z -3.8333, A 0.000, B 0.000, C 0.000 }
gfCNCPoint3[11557] = {X 337.8308, Y 30.8659, Z -3.8333, A 0.000, B 0.000, C 0.000 }
gfCNCPoint3[11558] = {X 338.2182, Y 31.5666, Z -3.8333, A 0.000, B 0.000, C 0.000 }
gfCNCPoint3[11559] = {X 338.4642, Y 32.3286, Z -3.8333, A 0.000, B 0.000, C 0.000 }
gfCNCPoint3[11560] = {X 338.5597, Y 33.1236, Z -3.8333, A 0.000, B 0.000, C 0.000 }
gfCNCPoint3[11561] = {X 338.5011, Y 33.9222, Z -3.8333, A 0.000, B 0.000, C 0.000 }
gfCNCPoint3[11562] = {X 339.2998, Y 34.6499, Z -3.8333, A 0.000, B 0.000, C 0.000 }
gfCNCPoint3[11563] = {X 340.1356, Y 35.3347, Z -3.8333, A 0.000, B 0.000, C 0.000 }
gfCNCPoint3[11564] = {X 341.4522, Y 36.1995, Z -3.8333, A 0.000, B 0.000, C 0.000 }
gfCNCPoint3[11565] = {X 342.8808, Y 36.8631, Z -3.8333, A 0.000, B 0.000, C 0.000 }
gfCNCPoint3[11566] = {X 344.3908, Y 37.3114, Z -3.8333, A 0.000, B 0.000, C 0.000 }
gfCNCPoint3[11567] = {X 345.9501, Y 37.5347, Z -3.8333, A 0.000, B 0.000, C 0.000 }
gfCNCPoint3[11568] = {X 347.5253, Y 37.5283, Z -3.8333, A 0.000, B 0.000, C 0.000 }
gfCNCPoint3[11569] = {X 348.7011, Y 37.3901, Z -3.8333, A 0.000, B 0.000, C 0.000 }
gfCNCPoint3[11570] = {X 349.8488, Y 37.0997, Z -3.8333, A 0.000, B 0.000, C 0.000 }
gfCNCPoint3[11571] = {X 350.9488, Y 36.6620, Z -3.8333, A 0.000, B 0.000, C 0.000 }
gfCNCPoint3[11572] = {X 351.9824, Y 36.0846, Z -3.8333, A 0.000, B 0.000, C 0.000 }
gfCNCPoint3[11573] = {X 352.9317, Y 35.3773, Z -3.8333, A 0.000, B 0.000, C 0.000 }
gfCNCPoint3[11574] = {X 354.1007, Y 34.2418, Z -3.8333, A 0.000, B 0.000, C 0.000 }
gfCNCPoint3[11575] = {X 355.1123, Y 32.9642, Z -3.8333, A 0.000, B 0.000, C 0.000 }
gfCNCPoint3[11576] = {X 355.9495, Y 31.5661, Z -3.8333, A 0.000, B 0.000, C 0.000 }
gfCNCPoint3[11577] = {X 356.5980, Y 30.0711, Z -3.8333, A 0.000, B 0.000, C 0.000 }
gfCNCPoint3[11578] = {X 357.0469, Y 28.5045, Z -3.8333, A 0.000, B 0.000, C 0.000 }
gfCNCPoint3[11579] = {X 357.3227, Y 26.8012, Z -3.8333, A 0.000, B 0.000, C 0.000 }
gfCNCPoint3[11580] = {X 357.4350, Y 25.0793, Z -3.8333, A 0.000, B 0.000, C 0.000 }
gfCNCPoint3[11581] = {X 357.3829, Y 23.3545, Z -3.8333, A 0.000, B 0.000, C 0.000 }
gfCNCPoint3[11582] = {X 357.1668, Y 21.6425, Z -3.8333, A 0.000, B 0.000, C 0.000 }
gfCNCPoint3[11583] = {X 356.8261, Y 20.1740, Z -3.8333, A 0.000, B 0.000, C 0.000 }
gfCNCPoint3[11584] = {X 356.3063, Y 18.7588, Z -3.8333, A 0.000, B 0.000, C 0.000 }
gfCNCPoint3[11585] = {X 355.6153, Y 17.4189, Z -3.8333, A 0.000, B 0.000, C 0.000 }
gfCNCPoint3[11586] = {X 354.7637, Y 16.1748, Z -3.8333, A 0.000, B 0.000, C 0.000 }
gfCNCPoint3[11587] = {X 353.8625, Y 15.1698, Z -3.8333, A 0.000, B 0.000, C 0.000 }
gfCNCPoint3[11588] = {X 352.8266, Y 14.3043, Z -3.8333, A 0.000, B 0.000, C 0.000 }
gfCNCPoint3[11589] = {X 351.6774, Y 13.5961, Z -3.8333, A 0.000, B 0.000, C 0.000 }
gfCNCPoint3[11590] = {X 350.4386, Y 13.0598, Z -3.8333, A 0.000, B 0.000, C 0.000 }
gfCNCPoint3[11591] = {X 349.1358, Y 12.7066, Z -3.8333, A 0.000, B 0.000, C 0.000 }
gfCNCPoint3[11592] = {X 347.5975, Y 12.5012, Z -3.8333, A 0.000, B 0.000, C 0.000 }
gfCNCPoint3[11593] = {X 346.0459, Y 12.4732, Z -3.8333, A 0.000, B 0.000, C 0.000 }
gfCNCPoint3[11594] = {X 344.5012, Y 12.6229, Z -3.8333, A 0.000, B 0.000, C 0.000 }
gfCNCPoint3[11595] = {X 342.9838, Y 12.9483, Z -3.8333, A 0.000, B 0.000, C 0.000 }
gfCNCPoint3[11596] = {X 341.5135, Y 13.4452, Z -3.8333, A 0.000, B 0.000, C 0.000 }
gfCNCPoint3[11597] = {X 340.1098, Y 14.1070, Z -3.8333, A 0.000, B 0.000, C 0.000 }
gfCNCPoint3[11598] = {X 338.7910, Y 14.9251, Z -3.8333, A 0.000, B 0.000, C 0.000 }
gfCNCPoint3[11599] = {X 338.7688, Y 15.7567, Z -3.8333, A 0.000, B 0.000, C 0.000 }
gfCNCPoint3[11600] = {X 338.5815, Y 16.5673, Z -3.8333, A 0.000, B 0.000, C 0.000 }
gfCNCPoint3[11601] = {X 338.2367, Y 17.3244, Z -3.8333, A 0.000, B 0.000, C 0.000 }
gfCNCPoint3[11602] = {X 337.7481, Y 17.9977, Z -3.8333, A 0.000, B 0.000, C 0.000 }
gfCNCPoint3[11603] = {X 337.1353, Y 18.5604, Z -3.8333, A 0.000, B 0.000, C 0.000 }
gfCNCPoint3[11604] = {X 336.4209, Y 19.0861, Z -3.8333, A 0.000, B 0.000, C 0.000 }
gfCNCPoint3[11605] = {X 335.6353, Y 19.5283, Z -3.8333, A 0.000, B 0.000, C 0.000 }
gfCNCPoint3[11606] = {X 334.7729, Y 19.7908, Z -3.8333, A 0.000, B 0.000, C 0.000 }
gfCNCPoint3[11607] = {X 333.8742, Y 19.8614, Z -3.8333, A 0.000, B 0.000, C 0.000 }
gfCNCPoint3[11608] = {X 332.9814, Y 19.7367, Z -3.8333, A 0.000, B 0.000, C 0.000 }
gfCNCPoint3[11609] = {X 332.1364, Y 19.4226, Z -3.8333, A 0.000, B 0.000, C 0.000 }
gfCNCPoint3[11610] = {X 331.3789, Y 18.9339, Z -3.8333, A 0.000, B 0.000, C 0.000 }
gfCNCPoint3[11611] = {X 330.7445, Y 18.2934, Z -3.8333, A 0.000, B 0.000, C 0.000 }
gfCNCPoint3[11612] = {X 330.2630, Y 17.5314, Z -3.8333, A 0.000, B 0.000, C 0.000 }
gfCNCPoint3[11613] = {X 326.7381, Y 10.2803, Z -3.8333, A 0.000, B 0.000, C 0.000 }
gfCNCPoint3[11614] = {X 326.4156, Y 9.3505, Z -3.8333, A 0.000, B 0.000, C 0.000 }
gfCNCPoint3[11615] = {X 326.3205, Y 8.3711, Z -3.8333, A 0.000, B 0.000, C 0.000 }
gfCNCPoint3[11616] = {X 326.4581, Y 7.3967, Z -3.8333, A 0.000, B 0.000, C 0.000 }
gfCNCPoint3[11617] = {X 326.8207, Y 6.4819, Z -3.8333, A 0.000, B 0.000, C 0.000 }
gfCNCPoint3[11618] = {X 327.3881, Y 5.6778, Z -3.8333, A 0.000, B 0.000, C 0.000 }
gfCNCPoint3[11619] = {X 328.1285, Y 5.0296, Z -3.8333, A 0.000, B 0.000, C 0.000 }
gfCNCPoint3[11620] = {X 328.7983, Y 4.5709, Z -3.8333, A 0.000, B 0.000, C 0.000 }
gfCNCPoint3[11621] = {X 329.6633, Y 4.1255, Z -3.8333, A 0.000, B 0.000, C 0.000 }
gfCNCPoint3[11622] = {X 330.6081, Y 3.8932, Z -3.8333, A 0.000, B 0.000, C 0.000 }
gfCNCPoint3[11623] = {X 331.5810, Y 3.8867, Z -3.8333, A 0.000, B 0.000, C 0.000 }
gfCNCPoint3[11624] = {X 332.5289, Y 4.1063, Z -3.8333, A 0.000, B 0.000, C 0.000 }
gfCNCPoint3[11625] = {X 334.0386, Y 3.2599, Z -3.8333, A 0.000, B 0.000, C 0.000 }
gfCNCPoint3[11626] = {X 335.5974, Y 2.5077, Z -3.8333, A 0.000, B 0.000, C 0.000 }
gfCNCPoint3[11627] = {X 337.7207, Y 1.6463, Z -3.8333, A 0.000, B 0.000, C 0.000 }
gfCNCPoint3[11628] = {X 339.9113, Y 0.9743, Z -3.8333, A 0.000, B 0.000, C 0.000 }
gfCNCPoint3[11629] = {X 342.1523, Y 0.4968, Z -3.8333, A 0.000, B 0.000, C 0.000 }
gfCNCPoint3[11630] = {X 344.4266, Y 0.2176, Z -3.8333, A 0.000, B 0.000, C 0.000 }
gfCNCPoint3[11631] = {X 346.7166, Y 0.1388, Z -3.8333, A 0.000, B 0.000, C 0.000 }
gfCNCPoint3[11632] = {X 349.0047, Y 0.2609, Z -3.8333, A 0.000, B 0.000, C 0.000 }
gfCNCPoint3[11633] = {X 351.2732, Y 0.5831, Z -3.8333, A 0.000, B 0.000, C 0.000 }
gfCNCPoint3[11634] = {X 351.5568, Y 0.6358, Z -3.8333, A 0.000, B 0.000, C 0.000 }
gfCNCPoint3[11635] = {X 352.2882, Y -3.2967, Z -3.8333, A 0.000, B 0.000, C 0.000 }
gfCNCPoint3[11636] = {X 351.5422, Y 0.7145, Z -3.8333, A 0.000, B 0.000, C 0.000 }
gfCNCPoint3[11637] = {X 351.8240, Y 0.7669, Z -3.8333, A 0.000, B 0.000, C 0.000 }
gfCNCPoint3[11638] = {X 353.7365, Y 1.2474, Z -3.8333, A 0.000, B 0.000, C 0.000 }
gfCNCPoint3[11639] = {X 355.5949, Y 1.9070, Z -3.8333, A 0.000, B 0.000, C 0.000 }
gfCNCPoint3[11640] = {X 357.3823, Y 2.7398, Z -3.8333, A 0.000, B 0.000, C 0.000 }
gfCNCPoint3[11641] = {X 359.0828, Y 3.7383, Z -3.8333, A 0.000, B 0.000, C 0.000 }
gfCNCPoint3[11642] = {X 360.6810, Y 4.8935, Z -3.8333, A 0.000, B 0.000, C 0.000 }
gfCNCPoint3[11643] = {X 362.1626, Y 6.1949, Z -3.8333, A 0.000, B 0.000, C 0.000 }
gfCNCPoint3[11644] = {X 363.5141, Y 7.6309, Z -3.8333, A 0.000, B 0.000, C 0.000 }
gfCNCPoint3[11645] = {X 364.9657, Y 9.5043, Z -3.8333, A 0.000, B 0.000, C 0.000 }
gfCNCPoint3[11646] = {X 366.2293, Y 11.5093, Z -3.8333, A 0.000, B 0.000, C 0.000 }
gfCNCPoint3[11647] = {X 367.2931, Y 13.6271, Z -3.8333, A 0.000, B 0.000, C 0.000 }
gfCNCPoint3[11648] = {X 368.1471, Y 15.8378, Z -3.8333, A 0.000, B 0.000, C 0.000 }
gfCNCPoint3[11649] = {X 368.7833, Y 18.1208, Z -3.8333, A 0.000, B 0.000, C 0.000 }
gfCNCPoint3[11650] = {X 369.2620, Y 20.7371, Z -3.8333, A 0.000, B 0.000, C 0.000 }
gfCNCPoint3[11651] = {X 369.5174, Y 23.3846, Z -3.8333, A 0.000, B 0.000, C 0.000 }
gfCNCPoint3[11652] = {X 369.5476, Y 26.0442, Z -3.8333, A 0.000, B 0.000, C 0.000 }
gfCNCPoint3[11653] = {X 369.3525, Y 28.6967, Z -3.8333, A 0.000, B 0.000, C 0.000 }
gfCNCPoint3[11654] = {X 368.9335, Y 31.3233, Z -3.8333, A 0.000, B 0.000, C 0.000 }
gfCNCPoint3[11655] = {X 368.4147, Y 33.4073, Z -3.8333, A 0.000, B 0.000, C 0.000 }
gfCNCPoint3[11656] = {X 367.7137, Y 35.4373, Z -3.8333, A 0.000, B 0.000, C 0.000 }
gfCNCPoint3[11657] = {X 366.8362, Y 37.3974, Z -3.8333, A 0.000, B 0.000, C 0.000 }
gfCNCPoint3[11658] = {X 365.7888, Y 39.2724, Z -3.8333, A 0.000, B 0.000, C 0.000 }
gfCNCPoint3[11659] = {X 364.5799, Y 41.0474, Z -3.8333, A 0.000, B 0.000, C 0.000 }
gfCNCPoint3[11660] = {X 364.4644, Y 41.2058, Z -3.8333, A 0.000, B 0.000, C 0.000 }
gfCNCPoint3[11661] = {X 363.8371, Y 41.9760, Z -3.8333, A 0.000, B 0.000, C 0.000 }
gfCNCPoint3[11662] = {X 362.5905, Y 43.3746, Z -3.8333, A 0.000, B 0.000, C 0.000 }
gfCNCPoint3[11663] = {X 361.2245, Y 44.6568, Z -3.8333, A 0.000, B 0.000, C 0.000 }
gfCNCPoint3[11664] = {X 359.7499, Y 45.8125, Z -3.8333, A 0.000, B 0.000, C 0.000 }
gfCNCPoint3[11665] = {X 358.1784, Y 46.8326, Z -3.8333, A 0.000, B 0.000, C 0.000 }
gfCNCPoint3[11666] = {X 356.5225, Y 47.7089, Z -3.8333, A 0.000, B 0.000, C 0.000 }
gfCNCPoint3[11667] = {X 356.1242, Y 47.8975, Z -3.8333, A 0.000, B 0.000, C 0.000 }
gfCNCPoint3[11668] = {X 353.9492, Y 48.7092, Z -3.8333, A 0.000, B 0.000, C 0.000 }
gfCNCPoint3[11669] = {X 351.7028, Y 49.2953, Z -3.8333, A 0.000, B 0.000, C 0.000 }
gfCNCPoint3[11670] = {X 349.4085, Y 49.6496, Z -3.8333, A 0.000, B 0.000, C 0.000 }
gfCNCPoint3[11671] = {X 347.0900, Y 49.7686, Z -3.8333, A 0.000, B 0.000, C 0.000 }
gfCNCPoint3[11672] = {X 345.0441, Y 49.7344, Z -3.8333, A 0.000, B 0.000, C 0.000 }
gfCNCPoint3[11673] = {X 343.0089, Y 49.5228, Z -3.8333, A 0.000, B 0.000, C 0.000 }
gfCNCPoint3[11674] = {X 340.9997, Y 49.1355, Z -3.8333, A 0.000, B 0.000, C 0.000 }
gfCNCPoint3[11675] = {X 339.0317, Y 48.5754, Z -3.8333, A 0.000, B 0.000, C 0.000 }
gfCNCPoint3[11676] = {X 337.1196, Y 47.8467, Z -3.8333, A 0.000, B 0.000, C 0.000 }
gfCNCPoint3[11677] = {X 335.2780, Y 46.9549, Z -3.8333, A 0.000, B 0.000, C 0.000 }
gfCNCPoint3[11678] = {X 333.6798, Y 45.9667, Z -3.8333, A 0.000, B 0.000, C 0.000 }
gfCNCPoint3[11679] = {X 332.1654, Y 44.8545, Z -3.8333, A 0.000, B 0.000, C 0.000 }
gfCNCPoint3[11680] = {X 330.7443, Y 43.6252, Z -3.8333, A 0.000, B 0.000, C 0.000 }
gfCNCPoint3[11681] = {X 329.8287, Y 43.6460, Z -3.8333, A 0.000, B 0.000, C 0.000 }
gfCNCPoint3[11682] = {X 328.9316, Y 43.4621, Z -3.8333, A 0.000, B 0.000, C 0.000 }
gfCNCPoint3[11683] = {X 328.0980, Y 43.0827, Z -3.8333, A 0.000, B 0.000, C 0.000 }
gfCNCPoint3[11684] = {X 327.3701, Y 42.5270, Z -3.8333, A 0.000, B 0.000, C 0.000 }
gfCNCPoint3[11685] = {X 326.7483, Y 41.9207, Z -3.8333, A 0.000, B 0.000, C 0.000 }
gfCNCPoint3[11686] = {X 326.1548, Y 41.1901, Z -3.8333, A 0.000, B 0.000, C 0.000 }
gfCNCPoint3[11687] = {X 325.7445, Y 40.3430, Z -3.8333, A 0.000, B 0.000, C 0.000 }
gfCNCPoint3[11688] = {X 325.5393, Y 39.4243, Z -3.8333, A 0.000, B 0.000, C 0.000 }
gfCNCPoint3[11689] = {X 325.5500, Y 38.4831, Z -3.8333, A 0.000, B 0.000, C 0.000 }
gfCNCPoint3[11690] = {X 325.7762, Y 37.5694, Z -3.8333, A 0.000, B 0.000, C 0.000 }
gfCNCPoint3[11691] = {X 326.2057, Y 36.7318, Z -3.8333, A 0.000, B 0.000, C 0.000 }
gfCNCPoint3[11692] = {X 330.4390, Y 30.4021, Z -3.8333, A 0.000, B 0.000, C 0.000 }
gfCNCPoint3[11693] = {X 331.0070, Y 29.7251, Z -3.8333, A 0.000, B 0.000, C 0.000 }
gfCNCPoint3[11694] = {X 331.7073, Y 29.1862, Z -3.8333, A 0.000, B 0.000, C 0.000 }
gfCNCPoint3[11695] = {X 332.5073, Y 28.8108, Z -3.8333, A 0.000, B 0.000, C 0.000 }
gfCNCPoint3[11696] = {X 333.3694, Y 28.6165, Z -3.8333, A 0.000, B 0.000, C 0.000 }
gfCNCPoint3[11697] = {X 334.2530, Y 28.6123, Z -3.8333, A 0.000, B 0.000, C 0.000 }
gfCNCPoint3[11698] = {X 335.1169, Y 28.7985, Z -3.8333, A 0.000, B 0.000, C 0.000 }
gfCNCPoint3[11699] = {X 335.9204, Y 29.1663, Z -3.8333, A 0.000, B 0.000, C 0.000 }
gfCNCPoint3[11700] = {X 336.6259, Y 29.6985, Z -3.8333, A 0.000, B 0.000, C 0.000 }
gfCNCPoint3[11701] = {X 337.2602, Y 30.3094, Z -3.8333, A 0.000, B 0.000, C 0.000 }
gfCNCPoint3[11702] = {X 337.7696, Y 30.9181, Z -3.8333, A 0.000, B 0.000, C 0.000 }
gfCNCPoint3[11703] = {X 338.1515, Y 31.6139, Z -3.8333, A 0.000, B 0.000, C 0.000 }
gfCNCPoint3[11704] = {X 338.3914, Y 32.3705, Z -3.8333, A 0.000, B 0.000, C 0.000 }
gfCNCPoint3[11705] = {X 338.4804, Y 33.1592, Z -3.8333, A 0.000, B 0.000, C 0.000 }
gfCNCPoint3[11706] = {X 338.4149, Y 33.9503, Z -3.8333, A 0.000, B 0.000, C 0.000 }
gfCNCPoint3[11707] = {X 339.2314, Y 34.6965, Z -3.8333, A 0.000, B 0.000, C 0.000 }
gfCNCPoint3[11708] = {X 340.0867, Y 35.3980, Z -3.8333, A 0.000, B 0.000, C 0.000 }
gfCNCPoint3[11709] = {X 341.4129, Y 36.2692, Z -3.8333, A 0.000, B 0.000, C 0.000 }
gfCNCPoint3[11710] = {X 342.8519, Y 36.9377, Z -3.8333, A 0.000, B 0.000, C 0.000 }
gfCNCPoint3[11711] = {X 344.3730, Y 37.3894, Z -3.8333, A 0.000, B 0.000, C 0.000 }
gfCNCPoint3[11712] = {X 345.9437, Y 37.6144, Z -3.8333, A 0.000, B 0.000, C 0.000 }
gfCNCPoint3[11713] = {X 347.5304, Y 37.6081, Z -3.8333, A 0.000, B 0.000, C 0.000 }
gfCNCPoint3[11714] = {X 348.7164, Y 37.4686, Z -3.8333, A 0.000, B 0.000, C 0.000 }
gfCNCPoint3[11715] = {X 349.8740, Y 37.1756, Z -3.8333, A 0.000, B 0.000, C 0.000 }
gfCNCPoint3[11716] = {X 350.9836, Y 36.7341, Z -3.8333, A 0.000, B 0.000, C 0.000 }
gfCNCPoint3[11717] = {X 352.0260, Y 36.1516, Z -3.8333, A 0.000, B 0.000, C 0.000 }
gfCNCPoint3[11718] = {X 352.9836, Y 35.4382, Z -3.8333, A 0.000, B 0.000, C 0.000 }
gfCNCPoint3[11719] = {X 354.1601, Y 34.2954, Z -3.8333, A 0.000, B 0.000, C 0.000 }
gfCNCPoint3[11720] = {X 355.1782, Y 33.0097, Z -3.8333, A 0.000, B 0.000, C 0.000 }
gfCNCPoint3[11721] = {X 356.0207, Y 31.6025, Z -3.8333, A 0.000, B 0.000, C 0.000 }
gfCNCPoint3[11722] = {X 356.6734, Y 30.0979, Z -3.8333, A 0.000, B 0.000, C 0.000 }
gfCNCPoint3[11723] = {X 357.1252, Y 28.5213, Z -3.8333, A 0.000, B 0.000, C 0.000 }
gfCNCPoint3[11724] = {X 357.4022, Y 26.8104, Z -3.8333, A 0.000, B 0.000, C 0.000 }
gfCNCPoint3[11725] = {X 357.5150, Y 25.0808, Z -3.8333, A 0.000, B 0.000, C 0.000 }
gfCNCPoint3[11726] = {X 357.4627, Y 23.3484, Z -3.8333, A 0.000, B 0.000, C 0.000 }
gfCNCPoint3[11727] = {X 357.2456, Y 21.6288, Z -3.8333, A 0.000, B 0.000, C 0.000 }
gfCNCPoint3[11728] = {X 356.9026, Y 20.1507, Z -3.8333, A 0.000, B 0.000, C 0.000 }
gfCNCPoint3[11729] = {X 356.3794, Y 18.7264, Z -3.8333, A 0.000, B 0.000, C 0.000 }
gfCNCPoint3[11730] = {X 355.6839, Y 17.3778, Z -3.8333, A 0.000, B 0.000, C 0.000 }
gfCNCPoint3[11731] = {X 354.8268, Y 16.1256, Z -3.8333, A 0.000, B 0.000, C 0.000 }
gfCNCPoint3[11732] = {X 353.9179, Y 15.1121, Z -3.8333, A 0.000, B 0.000, C 0.000 }
gfCNCPoint3[11733] = {X 352.8732, Y 14.2393, Z -3.8333, A 0.000, B 0.000, C 0.000 }
gfCNCPoint3[11734] = {X 351.7143, Y 13.5251, Z -3.8333, A 0.000, B 0.000, C 0.000 }
gfCNCPoint3[11735] = {X 350.4650, Y 12.9843, Z -3.8333, A 0.000, B 0.000, C 0.000 }
gfCNCPoint3[11736] = {X 349.1511, Y 12.6280, Z -3.8333, A 0.000, B 0.000, C 0.000 }
gfCNCPoint3[11737] = {X 347.5972, Y 12.4210, Z -3.8333, A 0.000, B 0.000, C 0.000 }
gfCNCPoint3[11738] = {X 346.0298, Y 12.3938, Z -3.8333, A 0.000, B 0.000, C 0.000 }
gfCNCPoint3[11739] = {X 344.4697, Y 12.5468, Z -3.8333, A 0.000, B 0.000, C 0.000 }
gfCNCPoint3[11740] = {X 342.9374, Y 12.8781, Z -3.8333, A 0.000, B 0.000, C 0.000 }
gfCNCPoint3[11741] = {X 341.4534, Y 13.3832, Z -3.8333, A 0.000, B 0.000, C 0.000 }
gfCNCPoint3[11742] = {X 340.0372, Y 14.0555, Z -3.8333, A 0.000, B 0.000, C 0.000 }
gfCNCPoint3[11743] = {X 338.7077, Y 14.8860, Z -3.8333, A 0.000, B 0.000, C 0.000 }
gfCNCPoint3[11744] = {X 338.6938, Y 15.7108, Z -3.8333, A 0.000, B 0.000, C 0.000 }
gfCNCPoint3[11745] = {X 338.5143, Y 16.5159, Z -3.8333, A 0.000, B 0.000, C 0.000 }
gfCNCPoint3[11746] = {X 338.1766, Y 17.2685, Z -3.8333, A 0.000, B 0.000, C 0.000 }
gfCNCPoint3[11747] = {X 337.6944, Y 17.9377, Z -3.8333, A 0.000, B 0.000, C 0.000 }
gfCNCPoint3[11748] = {X 337.0874, Y 18.4963, Z -3.8333, A 0.000, B 0.000, C 0.000 }
gfCNCPoint3[11749] = {X 336.3744, Y 19.0211, Z -3.8333, A 0.000, B 0.000, C 0.000 }
gfCNCPoint3[11750] = {X 335.6039, Y 19.4547, Z -3.8333, A 0.000, B 0.000, C 0.000 }
gfCNCPoint3[11751] = {X 334.7580, Y 19.7122, Z -3.8333, A 0.000, B 0.000, C 0.000 }
gfCNCPoint3[11752] = {X 333.8766, Y 19.7814, Z -3.8333, A 0.000, B 0.000, C 0.000 }
gfCNCPoint3[11753] = {X 333.0010, Y 19.6592, Z -3.8333, A 0.000, B 0.000, C 0.000 }
gfCNCPoint3[11754] = {X 332.1722, Y 19.3511, Z -3.8333, A 0.000, B 0.000, C 0.000 }
gfCNCPoint3[11755] = {X 331.4293, Y 18.8718, Z -3.8333, A 0.000, B 0.000, C 0.000 }
gfCNCPoint3[11756] = {X 330.8071, Y 18.2436, Z -3.8333, A 0.000, B 0.000, C 0.000 }
gfCNCPoint3[11757] = {X 330.3348, Y 17.4962, Z -3.8333, A 0.000, B 0.000, C 0.000 }
gfCNCPoint3[11758] = {X 326.8101, Y 10.2453, Z -3.8333, A 0.000, B 0.000, C 0.000 }
gfCNCPoint3[11759] = {X 326.4937, Y 9.3334, Z -3.8333, A 0.000, B 0.000, C 0.000 }
gfCNCPoint3[11760] = {X 326.4004, Y 8.3728, Z -3.8333, A 0.000, B 0.000, C 0.000 }
gfCNCPoint3[11761] = {X 326.5354, Y 7.4171, Z -3.8333, A 0.000, B 0.000, C 0.000 }
gfCNCPoint3[11762] = {X 326.8911, Y 6.5199, Z -3.8333, A 0.000, B 0.000, C 0.000 }
gfCNCPoint3[11763] = {X 327.4476, Y 5.7314, Z -3.8333, A 0.000, B 0.000, C 0.000 }
gfCNCPoint3[11764] = {X 328.1737, Y 5.0956, Z -3.8333, A 0.000, B 0.000, C 0.000 }
gfCNCPoint3[11765] = {X 328.8432, Y 4.6371, Z -3.8333, A 0.000, B 0.000, C 0.000 }
gfCNCPoint3[11766] = {X 329.7004, Y 4.1970, Z -3.8333, A 0.000, B 0.000, C 0.000 }
gfCNCPoint3[11767] = {X 330.6369, Y 3.9702, Z -3.8333, A 0.000, B 0.000, C 0.000 }
gfCNCPoint3[11768] = {X 331.6005, Y 3.9694, Z -3.8333, A 0.000, B 0.000, C 0.000 }
gfCNCPoint3[11769] = {X 332.5374, Y 4.1946, Z -3.8333, A 0.000, B 0.000, C 0.000 }
gfCNCPoint3[11770] = {X 334.0588, Y 3.3396, Z -3.8333, A 0.000, B 0.000, C 0.000 }
gfCNCPoint3[11771] = {X 335.6304, Y 2.5806, Z -3.8333, A 0.000, B 0.000, C 0.000 }
gfCNCPoint3[11772] = {X 337.7472, Y 1.7218, Z -3.8333, A 0.000, B 0.000, C 0.000 }
gfCNCPoint3[11773] = {X 339.9311, Y 1.0518, Z -3.8333, A 0.000, B 0.000, C 0.000 }
gfCNCPoint3[11774] = {X 342.1653, Y 0.5758, Z -3.8333, A 0.000, B 0.000, C 0.000 }
gfCNCPoint3[11775] = {X 344.4327, Y 0.2974, Z -3.8333, A 0.000, B 0.000, C 0.000 }
gfCNCPoint3[11776] = {X 346.7157, Y 0.2188, Z -3.8333, A 0.000, B 0.000, C 0.000 }
gfCNCPoint3[11777] = {X 348.9968, Y 0.3405, Z -3.8333, A 0.000, B 0.000, C 0.000 }
gfCNCPoint3[11778] = {X 351.2585, Y 0.6617, Z -3.8333, A 0.000, B 0.000, C 0.000 }
gfCNCPoint3[11779] = {X 351.5422, Y 0.7145, Z -3.8333, A 0.000, B 0.000, C 0.000 }
gfCNCPoint3[11780] = {X 352.2735, Y -3.2181, Z -3.8333, A 0.000, B 0.000, C 0.000 }
gfCNCPoint3[11781] = {X 351.5276, Y 0.7931, Z -3.8333, A 0.000, B 0.000, C 0.000 }
gfCNCPoint3[11782] = {X 351.8088, Y 0.8454, Z -3.8333, A 0.000, B 0.000, C 0.000 }
gfCNCPoint3[11783] = {X 353.7138, Y 1.3241, Z -3.8333, A 0.000, B 0.000, C 0.000 }
gfCNCPoint3[11784] = {X 355.5649, Y 1.9812, Z -3.8333, A 0.000, B 0.000, C 0.000 }
gfCNCPoint3[11785] = {X 357.3455, Y 2.8108, Z -3.8333, A 0.000, B 0.000, C 0.000 }
gfCNCPoint3[11786] = {X 359.0393, Y 3.8054, Z -3.8333, A 0.000, B 0.000, C 0.000 }
gfCNCPoint3[11787] = {X 360.6313, Y 4.9561, Z -3.8333, A 0.000, B 0.000, C 0.000 }
gfCNCPoint3[11788] = {X 362.1070, Y 6.2525, Z -3.8333, A 0.000, B 0.000, C 0.000 }
gfCNCPoint3[11789] = {X 363.4533, Y 7.6829, Z -3.8333, A 0.000, B 0.000, C 0.000 }
gfCNCPoint3[11790] = {X 364.9001, Y 9.5502, Z -3.8333, A 0.000, B 0.000, C 0.000 }
gfCNCPoint3[11791] = {X 366.1596, Y 11.5486, Z -3.8333, A 0.000, B 0.000, C 0.000 }
gfCNCPoint3[11792] = {X 367.2200, Y 13.6595, Z -3.8333, A 0.000, B 0.000, C 0.000 }
gfCNCPoint3[11793] = {X 368.0712, Y 15.8630, Z -3.8333, A 0.000, B 0.000, C 0.000 }
gfCNCPoint3[11794] = {X 368.7053, Y 18.1385, Z -3.8333, A 0.000, B 0.000, C 0.000 }
gfCNCPoint3[11795] = {X 369.1828, Y 20.7482, Z -3.8333, A 0.000, B 0.000, C 0.000 }
gfCNCPoint3[11796] = {X 369.4375, Y 23.3889, Z -3.8333, A 0.000, B 0.000, C 0.000 }
gfCNCPoint3[11797] = {X 369.4677, Y 26.0417, Z -3.8333, A 0.000, B 0.000, C 0.000 }
gfCNCPoint3[11798] = {X 369.2731, Y 28.6876, Z -3.8333, A 0.000, B 0.000, C 0.000 }
gfCNCPoint3[11799] = {X 368.8551, Y 31.3074, Z -3.8333, A 0.000, B 0.000, C 0.000 }
gfCNCPoint3[11800] = {X 368.3379, Y 33.3846, Z -3.8333, A 0.000, B 0.000, C 0.000 }
gfCNCPoint3[11801] = {X 367.6393, Y 35.4080, Z -3.8333, A 0.000, B 0.000, C 0.000 }
gfCNCPoint3[11802] = {X 366.7645, Y 37.3618, Z -3.8333, A 0.000, B 0.000, C 0.000 }
gfCNCPoint3[11803] = {X 365.7206, Y 39.2306, Z -3.8333, A 0.000, B 0.000, C 0.000 }
gfCNCPoint3[11804] = {X 364.5156, Y 40.9999, Z -3.8333, A 0.000, B 0.000, C 0.000 }
gfCNCPoint3[11805] = {X 364.4010, Y 41.1570, Z -3.8333, A 0.000, B 0.000, C 0.000 }
gfCNCPoint3[11806] = {X 363.7751, Y 41.9255, Z -3.8333, A 0.000, B 0.000, C 0.000 }
gfCNCPoint3[11807] = {X 362.5332, Y 43.3187, Z -3.8333, A 0.000, B 0.000, C 0.000 }
gfCNCPoint3[11808] = {X 361.1724, Y 44.5961, Z -3.8333, A 0.000, B 0.000, C 0.000 }
gfCNCPoint3[11809] = {X 359.7034, Y 45.7474, Z -3.8333, A 0.000, B 0.000, C 0.000 }
gfCNCPoint3[11810] = {X 358.1379, Y 46.7636, Z -3.8333, A 0.000, B 0.000, C 0.000 }
gfCNCPoint3[11811] = {X 356.4883, Y 47.6366, Z -3.8333, A 0.000, B 0.000, C 0.000 }
gfCNCPoint3[11812] = {X 356.0912, Y 47.8246, Z -3.8333, A 0.000, B 0.000, C 0.000 }
gfCNCPoint3[11813] = {X 353.9238, Y 48.6333, Z -3.8333, A 0.000, B 0.000, C 0.000 }
gfCNCPoint3[11814] = {X 351.6854, Y 49.2172, Z -3.8333, A 0.000, B 0.000, C 0.000 }
gfCNCPoint3[11815] = {X 349.3992, Y 49.5702, Z -3.8333, A 0.000, B 0.000, C 0.000 }
gfCNCPoint3[11816] = {X 347.0889, Y 49.6886, Z -3.8333, A 0.000, B 0.000, C 0.000 }
gfCNCPoint3[11817] = {X 345.0499, Y 49.6546, Z -3.8333, A 0.000, B 0.000, C 0.000 }
gfCNCPoint3[11818] = {X 343.0216, Y 49.4438, Z -3.8333, A 0.000, B 0.000, C 0.000 }
gfCNCPoint3[11819] = {X 341.0191, Y 49.0579, Z -3.8333, A 0.000, B 0.000, C 0.000 }
gfCNCPoint3[11820] = {X 339.0577, Y 48.4998, Z -3.8333, A 0.000, B 0.000, C 0.000 }
gfCNCPoint3[11821] = {X 337.1521, Y 47.7736, Z -3.8333, A 0.000, B 0.000, C 0.000 }
gfCNCPoint3[11822] = {X 335.3167, Y 46.8848, Z -3.8333, A 0.000, B 0.000, C 0.000 }
gfCNCPoint3[11823] = {X 333.7136, Y 45.8930, Z -3.8333, A 0.000, B 0.000, C 0.000 }
gfCNCPoint3[11824] = {X 332.1951, Y 44.7759, Z -3.8333, A 0.000, B 0.000, C 0.000 }
gfCNCPoint3[11825] = {X 330.7711, Y 43.5406, Z -3.8333, A 0.000, B 0.000, C 0.000 }
gfCNCPoint3[11826] = {X 329.8559, Y 43.5681, Z -3.8333, A 0.000, B 0.000, C 0.000 }
gfCNCPoint3[11827] = {X 328.9583, Y 43.3867, Z -3.8333, A 0.000, B 0.000, C 0.000 }
gfCNCPoint3[11828] = {X 328.1256, Y 43.0059, Z -3.8333, A 0.000, B 0.000, C 0.000 }
gfCNCPoint3[11829] = {X 327.4012, Y 42.4458, Z -3.8333, A 0.000, B 0.000, C 0.000 }
gfCNCPoint3[11830] = {X 326.8042, Y 41.8634, Z -3.8333, A 0.000, B 0.000, C 0.000 }
gfCNCPoint3[11831] = {X 326.2223, Y 41.1472, Z -3.8333, A 0.000, B 0.000, C 0.000 }
gfCNCPoint3[11832] = {X 325.8201, Y 40.3166, Z -3.8333, A 0.000, B 0.000, C 0.000 }
gfCNCPoint3[11833] = {X 325.6189, Y 39.4160, Z -3.8333, A 0.000, B 0.000, C 0.000 }
gfCNCPoint3[11834] = {X 325.6294, Y 38.4932, Z -3.8333, A 0.000, B 0.000, C 0.000 }
gfCNCPoint3[11835] = {X 325.8511, Y 37.5974, Z -3.8333, A 0.000, B 0.000, C 0.000 }
gfCNCPoint3[11836] = {X 326.2722, Y 36.7763, Z -3.8333, A 0.000, B 0.000, C 0.000 }
gfCNCPoint3[11837] = {X 330.5290, Y 30.4119, Z -3.8333, A 0.000, B 0.000, C 0.000 }
gfCNCPoint3[11838] = {X 331.0932, Y 29.7535, Z -3.8333, A 0.000, B 0.000, C 0.000 }
gfCNCPoint3[11839] = {X 331.7861, Y 29.2322, Z -3.8333, A 0.000, B 0.000, C 0.000 }
gfCNCPoint3[11840] = {X 332.5750, Y 28.8724, Z -3.8333, A 0.000, B 0.000, C 0.000 }
gfCNCPoint3[11841] = {X 333.4229, Y 28.6911, Z -3.8333, A 0.000, B 0.000, C 0.000 }
gfCNCPoint3[11842] = {X 334.2900, Y 28.6968, Z -3.8333, A 0.000, B 0.000, C 0.000 }
gfCNCPoint3[11843] = {X 335.1355, Y 28.8892, Z -3.8333, A 0.000, B 0.000, C 0.000 }
gfCNCPoint3[11844] = {X 335.9197, Y 29.2593, Z -3.8333, A 0.000, B 0.000, C 0.000 }
gfCNCPoint3[11845] = {X 336.6056, Y 29.7897, Z -3.8333, A 0.000, B 0.000, C 0.000 }
gfCNCPoint3[11846] = {X 337.2041, Y 30.3665, Z -3.8333, A 0.000, B 0.000, C 0.000 }
gfCNCPoint3[11847] = {X 337.7083, Y 30.9703, Z -3.8333, A 0.000, B 0.000, C 0.000 }
gfCNCPoint3[11848] = {X 338.0846, Y 31.6611, Z -3.8333, A 0.000, B 0.000, C 0.000 }
gfCNCPoint3[11849] = {X 338.3184, Y 32.4122, Z -3.8333, A 0.000, B 0.000, C 0.000 }
gfCNCPoint3[11850] = {X 338.4007, Y 33.1945, Z -3.8333, A 0.000, B 0.000, C 0.000 }
gfCNCPoint3[11851] = {X 338.3283, Y 33.9779, Z -3.8333, A 0.000, B 0.000, C 0.000 }
gfCNCPoint3[11852] = {X 339.1628, Y 34.7429, Z -3.8333, A 0.000, B 0.000, C 0.000 }
gfCNCPoint3[11853] = {X 340.0379, Y 35.4613, Z -3.8333, A 0.000, B 0.000, C 0.000 }
gfCNCPoint3[11854] = {X 341.2958, Y 36.2946, Z -3.8333, A 0.000, B 0.000, C 0.000 }
gfCNCPoint3[11855] = {X 342.6565, Y 36.9467, Z -3.8333, A 0.000, B 0.000, C 0.000 }
gfCNCPoint3[11856] = {X 344.0939, Y 37.4054, Z -3.8333, A 0.000, B 0.000, C 0.000 }
gfCNCPoint3[11857] = {X 345.5809, Y 37.6618, Z -3.8333, A 0.000, B 0.000, C 0.000 }
gfCNCPoint3[11858] = {X 347.0889, Y 37.7111, Z -3.8333, A 0.000, B 0.000, C 0.000 }
gfCNCPoint3[11859] = {X 347.5345, Y 37.6880, Z -3.8333, A 0.000, B 0.000, C 0.000 }
gfCNCPoint3[11860] = {X 348.7309, Y 37.5473, Z -3.8333, A 0.000, B 0.000, C 0.000 }
gfCNCPoint3[11861] = {X 349.8987, Y 37.2517, Z -3.8333, A 0.000, B 0.000, C 0.000 }
gfCNCPoint3[11862] = {X 351.0179, Y 36.8063, Z -3.8333, A 0.000, B 0.000, C 0.000 }
gfCNCPoint3[11863] = {X 352.0695, Y 36.2188, Z -3.8333, A 0.000, B 0.000, C 0.000 }
gfCNCPoint3[11864] = {X 353.0355, Y 35.4990, Z -3.8333, A 0.000, B 0.000, C 0.000 }
gfCNCPoint3[11865] = {X 354.2195, Y 34.3491, Z -3.8333, A 0.000, B 0.000, C 0.000 }
gfCNCPoint3[11866] = {X 355.2440, Y 33.0551, Z -3.8333, A 0.000, B 0.000, C 0.000 }
gfCNCPoint3[11867] = {X 356.0919, Y 31.6390, Z -3.8333, A 0.000, B 0.000, C 0.000 }
gfCNCPoint3[11868] = {X 356.7487, Y 30.1248, Z -3.8333, A 0.000, B 0.000, C 0.000 }
gfCNCPoint3[11869] = {X 357.2034, Y 28.5381, Z -3.8333, A 0.000, B 0.000, C 0.000 }
gfCNCPoint3[11870] = {X 357.4816, Y 26.8196, Z -3.8333, A 0.000, B 0.000, C 0.000 }
gfCNCPoint3[11871] = {X 357.5950, Y 25.0823, Z -3.8333, A 0.000, B 0.000, C 0.000 }
gfCNCPoint3[11872] = {X 357.5424, Y 23.3422, Z -3.8333, A 0.000, B 0.000, C 0.000 }
gfCNCPoint3[11873] = {X 357.3244, Y 21.6150, Z -3.8333, A 0.000, B 0.000, C 0.000 }
gfCNCPoint3[11874] = {X 356.9792, Y 20.1274, Z -3.8333, A 0.000, B 0.000, C 0.000 }
gfCNCPoint3[11875] = {X 356.4525, Y 18.6939, Z -3.8333, A 0.000, B 0.000, C 0.000 }
gfCNCPoint3[11876] = {X 355.7525, Y 17.3366, Z -3.8333, A 0.000, B 0.000, C 0.000 }
gfCNCPoint3[11877] = {X 354.8899, Y 16.0764, Z -3.8333, A 0.000, B 0.000, C 0.000 }
gfCNCPoint3[11878] = {X 353.9734, Y 15.0544, Z -3.8333, A 0.000, B 0.000, C 0.000 }
gfCNCPoint3[11879] = {X 352.9199, Y 14.1743, Z -3.8333, A 0.000, B 0.000, C 0.000 }
gfCNCPoint3[11880] = {X 351.7511, Y 13.4541, Z -3.8333, A 0.000, B 0.000, C 0.000 }
gfCNCPoint3[11881] = {X 350.4913, Y 12.9088, Z -3.8333, A 0.000, B 0.000, C 0.000 }
gfCNCPoint3[11882] = {X 349.1664, Y 12.5495, Z -3.8333, A 0.000, B 0.000, C 0.000 }
gfCNCPoint3[11883] = {X 347.3712, Y 12.3258, Z -3.8333, A 0.000, B 0.000, C 0.000 }
gfCNCPoint3[11884] = {X 345.5623, Y 12.3404, Z -3.8333, A 0.000, B 0.000, C 0.000 }
gfCNCPoint3[11885] = {X 343.7710, Y 12.5933, Z -3.8333, A 0.000, B 0.000, C 0.000 }
gfCNCPoint3[11886] = {X 342.0287, Y 13.0798, Z -3.8333, A 0.000, B 0.000, C 0.000 }
gfCNCPoint3[11887] = {X 340.3656, Y 13.7917, Z -3.8333, A 0.000, B 0.000, C 0.000 }
gfCNCPoint3[11888] = {X 338.8108, Y 14.7165, Z -3.8333, A 0.000, B 0.000, C 0.000 }
gfCNCPoint3[11889] = {X 338.7177, Y 14.7812, Z -3.8333, A 0.000, B 0.000, C 0.000 }
gfCNCPoint3[11890] = {X 338.6251, Y 14.8466, Z -3.8333, A 0.000, B 0.000, C 0.000 }
gfCNCPoint3[11891] = {X 338.6379, Y 15.0628, Z -3.8333, A 0.000, B 0.000, C 0.000 }
gfCNCPoint3[11892] = {X 338.5597, Y 16.0353, Z -3.8333, A 0.000, B 0.000, C 0.000 }
gfCNCPoint3[11893] = {X 338.2484, Y 16.9600, Z -3.8333, A 0.000, B 0.000, C 0.000 }
gfCNCPoint3[11894] = {X 337.7224, Y 17.7817, Z -3.8333, A 0.000, B 0.000, C 0.000 }
gfCNCPoint3[11895] = {X 337.0132, Y 18.4517, Z -3.8333, A 0.000, B 0.000, C 0.000 }
gfCNCPoint3[11896] = {X 336.3278, Y 18.9560, Z -3.8333, A 0.000, B 0.000, C 0.000 }
gfCNCPoint3[11897] = {X 335.5713, Y 19.3817, Z -3.8333, A 0.000, B 0.000, C 0.000 }
gfCNCPoint3[11898] = {X 334.7407, Y 19.6341, Z -3.8333, A 0.000, B 0.000, C 0.000 }
gfCNCPoint3[11899] = {X 333.8753, Y 19.7014, Z -3.8333, A 0.000, B 0.000, C 0.000 }
gfCNCPoint3[11900] = {X 333.0157, Y 19.5804, Z -3.8333, A 0.000, B 0.000, C 0.000 }
gfCNCPoint3[11901] = {X 332.2025, Y 19.2768, Z -3.8333, A 0.000, B 0.000, C 0.000 }
gfCNCPoint3[11902] = {X 331.4739, Y 18.8049, Z -3.8333, A 0.000, B 0.000, C 0.000 }
gfCNCPoint3[11903] = {X 330.8643, Y 18.1870, Z -3.8333, A 0.000, B 0.000, C 0.000 }
gfCNCPoint3[11904] = {X 330.4023, Y 17.4521, Z -3.8333, A 0.000, B 0.000, C 0.000 }
gfCNCPoint3[11905] = {X 326.8820, Y 10.2103, Z -3.8333, A 0.000, B 0.000, C 0.000 }
gfCNCPoint3[11906] = {X 326.5719, Y 9.3163, Z -3.8333, A 0.000, B 0.000, C 0.000 }
gfCNCPoint3[11907] = {X 326.4804, Y 8.3746, Z -3.8333, A 0.000, B 0.000, C 0.000 }
gfCNCPoint3[11908] = {X 326.6127, Y 7.4376, Z -3.8333, A 0.000, B 0.000, C 0.000 }
gfCNCPoint3[11909] = {X 326.9614, Y 6.5580, Z -3.8333, A 0.000, B 0.000, C 0.000 }
gfCNCPoint3[11910] = {X 327.5070, Y 5.7849, Z -3.8333, A 0.000, B 0.000, C 0.000 }
gfCNCPoint3[11911] = {X 328.2189, Y 5.1616, Z -3.8333, A 0.000, B 0.000, C 0.000 }
gfCNCPoint3[11912] = {X 328.8880, Y 4.7034, Z -3.8333, A 0.000, B 0.000, C 0.000 }
gfCNCPoint3[11913] = {X 329.7043, Y 4.2813, Z -3.8333, A 0.000, B 0.000, C 0.000 }
gfCNCPoint3[11914] = {X 330.5954, Y 4.0567, Z -3.8333, A 0.000, B 0.000, C 0.000 }
gfCNCPoint3[11915] = {X 331.5142, Y 4.0413, Z -3.8333, A 0.000, B 0.000, C 0.000 }
gfCNCPoint3[11916] = {X 332.4122, Y 4.2361, Z -3.8333, A 0.000, B 0.000, C 0.000 }
gfCNCPoint3[11917] = {X 332.5467, Y 4.2824, Z -3.8333, A 0.000, B 0.000, C 0.000 }
gfCNCPoint3[11918] = {X 332.6259, Y 4.2347, Z -3.8333, A 0.000, B 0.000, C 0.000 }
gfCNCPoint3[11919] = {X 332.7051, Y 4.1872, Z -3.8333, A 0.000, B 0.000, C 0.000 }
gfCNCPoint3[11920] = {X 334.1612, Y 3.3765, Z -3.8333, A 0.000, B 0.000, C 0.000 }
gfCNCPoint3[11921] = {X 335.6629, Y 2.6537, Z -3.8333, A 0.000, B 0.000, C 0.000 }
gfCNCPoint3[11922] = {X 336.0092, Y 2.4996, Z -3.8333, A 0.000, B 0.000, C 0.000 }
gfCNCPoint3[11923] = {X 338.0805, Y 1.6915, Z -3.8333, A 0.000, B 0.000, C 0.000 }
gfCNCPoint3[11924] = {X 340.2133, Y 1.0636, Z -3.8333, A 0.000, B 0.000, C 0.000 }
gfCNCPoint3[11925] = {X 342.3920, Y 0.6205, Z -3.8333, A 0.000, B 0.000, C 0.000 }
gfCNCPoint3[11926] = {X 344.6007, Y 0.3655, Z -3.8333, A 0.000, B 0.000, C 0.000 }
gfCNCPoint3[11927] = {X 346.8231, Y 0.3004, Z -3.8333, A 0.000, B 0.000, C 0.000 }
gfCNCPoint3[11928] = {X 349.0429, Y 0.4256, Z -3.8333, A 0.000, B 0.000, C 0.000 }
gfCNCPoint3[11929] = {X 351.2438, Y 0.7404, Z -3.8333, A 0.000, B 0.000, C 0.000 }
gfCNCPoint3[11930] = {X 351.5276, Y 0.7931, Z -3.8333, A 0.000, B 0.000, C 0.000 }
gfCNCPoint3[11931] = {X 352.2735, Y -3.2181, Z -3.8333, A 0.000, B 0.000, C 0.000 }
gfCNCPoint3[11932] = {X 352.2735, Y -3.2181, Z -0.8333, A 0.000, B 0.000, C 0.000 }
gfCNCPoint3[11933] = {X 352.2735, Y -3.2181, Z 11.0000, A 0.000, B 0.000, C 0.000 }
gfCNCPoint3[11934] = {X 606.0427, Y 42.9009, Z 11.0000, A 0.000, B 0.000, C 0.000 }
gfCNCPoint3[11935] = {X 606.0427, Y 42.9009, Z -0.8333, A 0.000, B 0.000, C 0.000 }
gfCNCPoint3[11936] = {X 606.0427, Y 42.9009, Z -3.8333, A 0.000, B 0.000, C 0.000 }
gfCNCPoint3[11937] = {X 603.6965, Y 47.0768, Z -3.8333, A 0.000, B 0.000, C 0.000 }
gfCNCPoint3[11938] = {X 603.6310, Y 47.1893, Z -3.8333, A 0.000, B 0.000, C 0.000 }
gfCNCPoint3[11939] = {X 603.5621, Y 47.2998, Z -3.8333, A 0.000, B 0.000, C 0.000 }
gfCNCPoint3[11940] = {X 603.0357, Y 47.9601, Z -3.8333, A 0.000, B 0.000, C 0.000 }
gfCNCPoint3[11941] = {X 602.3889, Y 48.5030, Z -3.8333, A 0.000, B 0.000, C 0.000 }
gfCNCPoint3[11942] = {X 601.6472, Y 48.9069, Z -3.8333, A 0.000, B 0.000, C 0.000 }
gfCNCPoint3[11943] = {X 600.8403, Y 49.1559, Z -3.8333, A 0.000, B 0.000, C 0.000 }
gfCNCPoint3[11944] = {X 600.0000, Y 49.2400, Z -3.8333, A 0.000, B 0.000, C 0.000 }
gfCNCPoint3[11945] = {X 593.5565, Y 49.2400, Z -3.8333, A 0.000, B 0.000, C 0.000 }
gfCNCPoint3[11946] = {X 592.6130, Y 49.1337, Z -3.8333, A 0.000, B 0.000, C 0.000 }
gfCNCPoint3[11947] = {X 591.7169, Y 48.8201, Z -3.8333, A 0.000, B 0.000, C 0.000 }
gfCNCPoint3[11948] = {X 590.9129, Y 48.3150, Z -3.8333, A 0.000, B 0.000, C 0.000 }
gfCNCPoint3[11949] = {X 590.2416, Y 47.6436, Z -3.8333, A 0.000, B 0.000, C 0.000 }
gfCNCPoint3[11950] = {X 589.7364, Y 46.8397, Z -3.8333, A 0.000, B 0.000, C 0.000 }
gfCNCPoint3[11951] = {X 589.4228, Y 45.9435, Z -3.8333, A 0.000, B 0.000, C 0.000 }
gfCNCPoint3[11952] = {X 589.3165, Y 45.0000, Z -3.8333, A 0.000, B 0.000, C 0.000 }
gfCNCPoint3[11953] = {X 589.3165, Y 44.0649, Z -3.8333, A 0.000, B 0.000, C 0.000 }
gfCNCPoint3[11954] = {X 589.4211, Y 43.1447, Z -3.8333, A 0.000, B 0.000, C 0.000 }
gfCNCPoint3[11955] = {X 589.7210, Y 42.2686, Z -3.8333, A 0.000, B 0.000, C 0.000 }
gfCNCPoint3[11956] = {X 590.2023, Y 41.4775, Z -3.8333, A 0.000, B 0.000, C 0.000 }
gfCNCPoint3[11957] = {X 590.8425, Y 40.8084, Z -3.8333, A 0.000, B 0.000, C 0.000 }
gfCNCPoint3[11958] = {X 590.8430, Y 33.1200, Z -3.8333, A 0.000, B 0.000, C 0.000 }
gfCNCPoint3[11959] = {X 585.3714, Y 46.6218, Z -3.8333, A 0.000, B 0.000, C 0.000 }
gfCNCPoint3[11960] = {X 585.0085, Y 47.3114, Z -3.8333, A 0.000, B 0.000, C 0.000 }
gfCNCPoint3[11961] = {X 584.5255, Y 47.9228, Z -3.8333, A 0.000, B 0.000, C 0.000 }
gfCNCPoint3[11962] = {X 583.9387, Y 48.4356, Z -3.8333, A 0.000, B 0.000, C 0.000 }
gfCNCPoint3[11963] = {X 583.2680, Y 48.8323, Z -3.8333, A 0.000, B 0.000, C 0.000 }
gfCNCPoint3[11964] = {X 582.3418, Y 49.1460, Z -3.8333, A 0.000, B 0.000, C 0.000 }
gfCNCPoint3[11965] = {X 581.3682, Y 49.2391, Z -3.8333, A 0.000, B 0.000, C 0.000 }
gfCNCPoint3[11966] = {X 580.3993, Y 49.1068, Z -3.8333, A 0.000, B 0.000, C 0.000 }
gfCNCPoint3[11967] = {X 579.4864, Y 48.7559, Z -3.8333, A 0.000, B 0.000, C 0.000 }
gfCNCPoint3[11968] = {X 578.6782, Y 48.2052, Z -3.8333, A 0.000, B 0.000, C 0.000 }
gfCNCPoint3[11969] = {X 578.0177, Y 47.4840, Z -3.8333, A 0.000, B 0.000, C 0.000 }
gfCNCPoint3[11970] = {X 577.5400, Y 46.6307, Z -3.8333, A 0.000, B 0.000, C 0.000 }
gfCNCPoint3[11971] = {X 571.9386, Y 32.9337, Z -3.8333, A 0.000, B 0.000, C 0.000 }
gfCNCPoint3[11972] = {X 571.9389, Y 40.8080, Z -3.8333, A 0.000, B 0.000, C 0.000 }
gfCNCPoint3[11973] = {X 571.9706, Y 40.8338, Z -3.8333, A 0.000, B 0.000, C 0.000 }
gfCNCPoint3[11974] = {X 572.5959, Y 41.4922, Z -3.8333, A 0.000, B 0.000, C 0.000 }
gfCNCPoint3[11975] = {X 573.0667, Y 42.2686, Z -3.8333, A 0.000, B 0.000, C 0.000 }
gfCNCPoint3[11976] = {X 573.3613, Y 43.1275, Z -3.8333, A 0.000, B 0.000, C 0.000 }
gfCNCPoint3[11977] = {X 573.4663, Y 44.0294, Z -3.8333, A 0.000, B 0.000, C 0.000 }
gfCNCPoint3[11978] = {X 573.4664, Y 45.0000, Z -3.8333, A 0.000, B 0.000, C 0.000 }
gfCNCPoint3[11979] = {X 573.3601, Y 45.9435, Z -3.8333, A 0.000, B 0.000, C 0.000 }
gfCNCPoint3[11980] = {X 573.0465, Y 46.8397, Z -3.8333, A 0.000, B 0.000, C 0.000 }
gfCNCPoint3[11981] = {X 572.5414, Y 47.6436, Z -3.8333, A 0.000, B 0.000, C 0.000 }
gfCNCPoint3[11982] = {X 571.8700, Y 48.3150, Z -3.8333, A 0.000, B 0.000, C 0.000 }
gfCNCPoint3[11983] = {X 571.0661, Y 48.8201, Z -3.8333, A 0.000, B 0.000, C 0.000 }
gfCNCPoint3[11984] = {X 570.1699, Y 49.1337, Z -3.8333, A 0.000, B 0.000, C 0.000 }
gfCNCPoint3[11985] = {X 569.2264, Y 49.2400, Z -3.8333, A 0.000, B 0.000, C 0.000 }
gfCNCPoint3[11986] = {X 562.4443, Y 49.2400, Z -3.8333, A 0.000, B 0.000, C 0.000 }
gfCNCPoint3[11987] = {X 561.5008, Y 49.1337, Z -3.8333, A 0.000, B 0.000, C 0.000 }
gfCNCPoint3[11988] = {X 560.6046, Y 48.8201, Z -3.8333, A 0.000, B 0.000, C 0.000 }
gfCNCPoint3[11989] = {X 559.8007, Y 48.3150, Z -3.8333, A 0.000, B 0.000, C 0.000 }
gfCNCPoint3[11990] = {X 559.1293, Y 47.6436, Z -3.8333, A 0.000, B 0.000, C 0.000 }
gfCNCPoint3[11991] = {X 558.6242, Y 46.8397, Z -3.8333, A 0.000, B 0.000, C 0.000 }
gfCNCPoint3[11992] = {X 558.3106, Y 45.9435, Z -3.8333, A 0.000, B 0.000, C 0.000 }
gfCNCPoint3[11993] = {X 558.2043, Y 45.0000, Z -3.8333, A 0.000, B 0.000, C 0.000 }
gfCNCPoint3[11994] = {X 558.2043, Y 44.0650, Z -3.8333, A 0.000, B 0.000, C 0.000 }
gfCNCPoint3[11995] = {X 558.3087, Y 43.1444, Z -3.8333, A 0.000, B 0.000, C 0.000 }
gfCNCPoint3[11996] = {X 558.6089, Y 42.2680, Z -3.8333, A 0.000, B 0.000, C 0.000 }
gfCNCPoint3[11997] = {X 559.0909, Y 41.4769, Z -3.8333, A 0.000, B 0.000, C 0.000 }
gfCNCPoint3[11998] = {X 559.7321, Y 40.8081, Z -3.8333, A 0.000, B 0.000, C 0.000 }
gfCNCPoint3[11999] = {X 559.7321, Y 9.1931, Z -3.8333, A 0.000, B 0.000, C 0.000 }
gfCNCPoint3[12000] = {X 559.0940, Y 8.5328, Z -3.8333, A 0.000, B 0.000, C 0.000 }
gfCNCPoint3[12001] = {X 558.6131, Y 7.7505, Z -3.8333, A 0.000, B 0.000, C 0.000 }
gfCNCPoint3[12002] = {X 558.3119, Y 6.8831, Z -3.8333, A 0.000, B 0.000, C 0.000 }
gfCNCPoint3[12003] = {X 558.2045, Y 5.9711, Z -3.8333, A 0.000, B 0.000, C 0.000 }
gfCNCPoint3[12004] = {X 558.2043, Y 5.0000, Z -3.8333, A 0.000, B 0.000, C 0.000 }
gfCNCPoint3[12005] = {X 558.3106, Y 4.0565, Z -3.8333, A 0.000, B 0.000, C 0.000 }
gfCNCPoint3[12006] = {X 558.6242, Y 3.1603, Z -3.8333, A 0.000, B 0.000, C 0.000 }
gfCNCPoint3[12007] = {X 559.1293, Y 2.3564, Z -3.8333, A 0.000, B 0.000, C 0.000 }
gfCNCPoint3[12008] = {X 559.8007, Y 1.6850, Z -3.8333, A 0.000, B 0.000, C 0.000 }
gfCNCPoint3[12009] = {X 560.6046, Y 1.1799, Z -3.8333, A 0.000, B 0.000, C 0.000 }
gfCNCPoint3[12010] = {X 561.5008, Y 0.8663, Z -3.8333, A 0.000, B 0.000, C 0.000 }
gfCNCPoint3[12011] = {X 562.4443, Y 0.7600, Z -3.8333, A 0.000, B 0.000, C 0.000 }
gfCNCPoint3[12012] = {X 570.9376, Y 0.7600, Z -3.8333, A 0.000, B 0.000, C 0.000 }
gfCNCPoint3[12013] = {X 571.8810, Y 0.8663, Z -3.8333, A 0.000, B 0.000, C 0.000 }
gfCNCPoint3[12014] = {X 572.7772, Y 1.1799, Z -3.8333, A 0.000, B 0.000, C 0.000 }
gfCNCPoint3[12015] = {X 573.5812, Y 1.6850, Z -3.8333, A 0.000, B 0.000, C 0.000 }
gfCNCPoint3[12016] = {X 574.2525, Y 2.3564, Z -3.8333, A 0.000, B 0.000, C 0.000 }
gfCNCPoint3[12017] = {X 574.7577, Y 3.1603, Z -3.8333, A 0.000, B 0.000, C 0.000 }
gfCNCPoint3[12018] = {X 575.0712, Y 4.0565, Z -3.8333, A 0.000, B 0.000, C 0.000 }
gfCNCPoint3[12019] = {X 575.1776, Y 5.0000, Z -3.8333, A 0.000, B 0.000, C 0.000 }
gfCNCPoint3[12020] = {X 575.1776, Y 5.9342, Z -3.8333, A 0.000, B 0.000, C 0.000 }
gfCNCPoint3[12021] = {X 575.1023, Y 6.7292, Z -3.8333, A 0.000, B 0.000, C 0.000 }
gfCNCPoint3[12022] = {X 574.8794, Y 7.4960, Z -3.8333, A 0.000, B 0.000, C 0.000 }
gfCNCPoint3[12023] = {X 574.5166, Y 8.2074, Z -3.8333, A 0.000, B 0.000, C 0.000 }
gfCNCPoint3[12024] = {X 581.1908, Y 24.5818, Z -3.8333, A 0.000, B 0.000, C 0.000 }
gfCNCPoint3[12025] = {X 587.9348, Y 8.0880, Z -3.8333, A 0.000, B 0.000, C 0.000 }
gfCNCPoint3[12026] = {X 587.6159, Y 7.4200, Z -3.8333, A 0.000, B 0.000, C 0.000 }
gfCNCPoint3[12027] = {X 587.4179, Y 6.7067, Z -3.8333, A 0.000, B 0.000, C 0.000 }
gfCNCPoint3[12028] = {X 587.3471, Y 5.9698, Z -3.8333, A 0.000, B 0.000, C 0.000 }
gfCNCPoint3[12029] = {X 587.3470, Y 5.0000, Z -3.8333, A 0.000, B 0.000, C 0.000 }
gfCNCPoint3[12030] = {X 587.4533, Y 4.0565, Z -3.8333, A 0.000, B 0.000, C 0.000 }
gfCNCPoint3[12031] = {X 587.7668, Y 3.1603, Z -3.8333, A 0.000, B 0.000, C 0.000 }
gfCNCPoint3[12032] = {X 588.2720, Y 2.3564, Z -3.8333, A 0.000, B 0.000, C 0.000 }
gfCNCPoint3[12033] = {X 588.9434, Y 1.6850, Z -3.8333, A 0.000, B 0.000, C 0.000 }
gfCNCPoint3[12034] = {X 589.7473, Y 1.1799, Z -3.8333, A 0.000, B 0.000, C 0.000 }
gfCNCPoint3[12035] = {X 590.6435, Y 0.8663, Z -3.8333, A 0.000, B 0.000, C 0.000 }
gfCNCPoint3[12036] = {X 591.5870, Y 0.7600, Z -3.8333, A 0.000, B 0.000, C 0.000 }
gfCNCPoint3[12037] = {X 600.0000, Y 0.7600, Z -3.8333, A 0.000, B 0.000, C 0.000 }
gfCNCPoint3[12038] = {X 600.8403, Y 0.8441, Z -3.8333, A 0.000, B 0.000, C 0.000 }
gfCNCPoint3[12039] = {X 601.6472, Y 1.0931, Z -3.8333, A 0.000, B 0.000, C 0.000 }
gfCNCPoint3[12040] = {X 602.3889, Y 1.4970, Z -3.8333, A 0.000, B 0.000, C 0.000 }
gfCNCPoint3[12041] = {X 603.0357, Y 2.0399, Z -3.8333, A 0.000, B 0.000, C 0.000 }
gfCNCPoint3[12042] = {X 603.5621, Y 2.7002, Z -3.8333, A 0.000, B 0.000, C 0.000 }
gfCNCPoint3[12043] = {X 603.6310, Y 2.8107, Z -3.8333, A 0.000, B 0.000, C 0.000 }
gfCNCPoint3[12044] = {X 603.6965, Y 2.9232, Z -3.8333, A 0.000, B 0.000, C 0.000 }
gfCNCPoint3[12045] = {X 607.8231, Y 10.2681, Z -3.8333, A 0.000, B 0.000, C 0.000 }
gfCNCPoint3[12046] = {X 607.8231, Y 10.2681, Z -0.8333, A 0.000, B 0.000, C 0.000 }
gfCNCPoint3[12047] = {X 607.8231, Y 10.2681, Z 11.0000, A 0.000, B 0.000, C 0.000 }
gfCNCPoint3[12048] = {X 607.6965, Y 39.1593, Z 11.0000, A 0.000, B 0.000, C 0.000 }
gfCNCPoint3[12049] = {X 607.6965, Y 39.1593, Z -0.8333, A 0.000, B 0.000, C 0.000 }
gfCNCPoint3[12050] = {X 607.6965, Y 39.1593, Z -3.8333, A 0.000, B 0.000, C 0.000 }
gfCNCPoint3[12051] = {X 603.6965, Y 46.9082, Z -3.8333, A 0.000, B 0.000, C 0.000 }
gfCNCPoint3[12052] = {X 603.5999, Y 47.0847, Z -3.8333, A 0.000, B 0.000, C 0.000 }
gfCNCPoint3[12053] = {X 603.4949, Y 47.2564, Z -3.8333, A 0.000, B 0.000, C 0.000 }
gfCNCPoint3[12054] = {X 602.9784, Y 47.9042, Z -3.8333, A 0.000, B 0.000, C 0.000 }
gfCNCPoint3[12055] = {X 602.3438, Y 48.4369, Z -3.8333, A 0.000, B 0.000, C 0.000 }
gfCNCPoint3[12056] = {X 601.6162, Y 48.8332, Z -3.8333, A 0.000, B 0.000, C 0.000 }
gfCNCPoint3[12057] = {X 600.8244, Y 49.0775, Z -3.8333, A 0.000, B 0.000, C 0.000 }
gfCNCPoint3[12058] = {X 600.0000, Y 49.1600, Z -3.8333, A 0.000, B 0.000, C 0.000 }
gfCNCPoint3[12059] = {X 593.5565, Y 49.1600, Z -3.8333, A 0.000, B 0.000, C 0.000 }
gfCNCPoint3[12060] = {X 592.6308, Y 49.0557, Z -3.8333, A 0.000, B 0.000, C 0.000 }
gfCNCPoint3[12061] = {X 591.7516, Y 48.7480, Z -3.8333, A 0.000, B 0.000, C 0.000 }
gfCNCPoint3[12062] = {X 590.9628, Y 48.2524, Z -3.8333, A 0.000, B 0.000, C 0.000 }
gfCNCPoint3[12063] = {X 590.3041, Y 47.5937, Z -3.8333, A 0.000, B 0.000, C 0.000 }
gfCNCPoint3[12064] = {X 589.8085, Y 46.8050, Z -3.8333, A 0.000, B 0.000, C 0.000 }
gfCNCPoint3[12065] = {X 589.5008, Y 45.9257, Z -3.8333, A 0.000, B 0.000, C 0.000 }
gfCNCPoint3[12066] = {X 589.3965, Y 45.0000, Z -3.8333, A 0.000, B 0.000, C 0.000 }
